// TIA Portal V16 export
// export: Created 2021-03-19T14:27:15.418879Z, ExportSetting WithDefaults, DisplayName Totally Integrated Automation Portal, DisplayVersion V16 Update 3, DisplayName TIA Portal Version Control Interface, DisplayVersion V16 Update 2, DisplayName TIA Portal Openness, DisplayVersion V16 Update 3, DisplayName STEP 7 Professional, DisplayVersion V16 Update 3, DisplayName STEP 7 Safety, DisplayVersion V16, DisplayName WinCC Professional, DisplayVersion V16 Update 3
FUNCTION "FC02001_StdInstAnalogRead" : Void   // FC2001, LAD
TITLE = Standard - Inst — Analog Instrument Read and Scale
{ S7_Optimized_Access := 'TRUE' }
AUTHOR : M_Gledhill
FAMILY : Instrumentation
NAME : StdInstAnalogRead
VERSION : 1.0
// PRACTICAL SERIES AUTOMATION LIBRARY (PAL)   —   COPYRIGHT 2020 – M. GLEDHILL (MIT LICENCE)
//                   ———— ◆ ————
//  FOR DETAILED DOCUMENTATION — SELECT THE BLOCK IN THE PROJECT TREE AND PRESS SHIFT + F1
//  FULL ONLINE DOCUMENTATION IS AVAILABLE AT: https://practicalseries.com/2001-pal/index.html
// stored: AutoNumber false, IsIECCheckEnabled false, SetENOAutomatically false, UDAEnableTagReadback false
   VAR_INPUT
      SYS_SIGNALS : "UT21000_Dy_SysSignals";   // Common system signals — logic and timing signals
      RAW_ANALOG : Int;   // Analogue Input Signal
      EXT_FAULT : Bool;   // Instrument External Fault (1 = Fault, 0 = Healthy)
   END_VAR
   VAR_IN_OUT
      STATIC_DATA : "UT02001_St_InstAnalogRead";   // Static data storage (UDT)
      DYNAMIC_DATA : "UT22001_Dy_InstAnalogRead";   // Dynamic data storage (UDT)
   END_VAR
   VAR_TEMP
      revInfo : "UT01000_St_SysRevision";   // Revision information for this block
      licInfo : "UT01001_St_SysLicence";   // Licence information for this block
      wrkAlmHEn : Bool;   // Working storage (Alm_H is enabled and not masked)
      wrkAlmLEn : Bool;   // Working storage (Alm_L is enabled and not masked)
      wrkWrnHEn : Bool;   // Working storage (Wrn_H is enabled and not masked)
      wrkWrnLEn : Bool;   // Working storage (Wrn_L is enabled and not masked)
      calcPart1 : Real;   // Scale value calculation part 1 (RAW_VALUE − RAW_MIN)
      calcPart2 : Real;   // Scale value calculation part 2 (SCALE_MAX − SCALE_MIN)
      calcPart3 : Real;   // Scale value calculation part 1 (RAW_MAX − RAW_MIN)
      calcRawOOR : Real;   // Calculated OOR absolute value in terms of the RAW_VALUE
      calcOverRange : Real;   // Calculated over range limit (in raw units)
      calcUnderRange : Real;   // Calculated under range limit (in raw units)
      calcHystAbs : Real;   // Absolute Hysteresis (in relation to alarm/waringin)
      wrkHyst : Real;   // Working hysteresis value
      wrkOORPercent : Real;   // Working out of range percentage
      wrkInt : Int;   // Working storage (Integer)
      wrkReal : Real;   // Working storage (real)
      wrkDInt : DInt;   // Working storage (Double integer)
   END_VAR
   VAR_TEMP   // added for the SCL form of the ladder/FBD networks
      _w1 : Bool;
      _w2 : Bool;
      _w3 : Bool;
      _w4 : Bool;
   END_VAR
BEGIN

REGION Network 1: Block description — Sections 1 to 3.1
   // ▀▀▀▀▀▀▀▀▀▀▀▀▀▀▀▀▀▀▀▀▀▀▀▀▀▀▀▀▀▀▀▀▀▀▀▀▀▀▀▀▀▀▀▀
   // 
   // TITLE:    STANDARD ANALOG INSTRUMENT READ, SCALE AND ALARM MONITORING
   // 
   // ▄▄▄▄▄▄▄▄▄▄▄▄▄▄▄▄▄▄▄▄▄▄▄▄▄▄▄▄▄▄▄▄▄▄▄▄▄▄▄▄▄▄▄▄
   // 
   // 
   // 
   // This block reads and scales an analogue instrument signal received via an analogue input card.
   // 
   // The resultant scaled value is a real (floating point) number that matches the calibrated range of 
   // the instrument in engineering units.
   // 
   // The block has the facility to generate up to four alarms and warnings whenever the signal is 
   // beyond a specific setpoint value (either above or below); the four signals are:
   // 
   //    •   Alarm high
   // 
   //    •   Warning high
   // 
   //    •   Warning low
   // 
   //    •   Alarm low
   // 
   // Each alarm or warning can be time filtered (the condition must be present for a preset time 
   // before the alarm or warning is activated) and each will automatically reset when the signal is 
   // back within the acceptable range by a hysteresis amount.
   // 
   // In addition to the above four signals, various out-of-range fault signals will be generated if the 
   // instrument is outside its normal calibrated range by more than a specified percentage (this 
   // being a percentage of the total span of the instruments range).
   // 
   // The block can also generate an optional “external fault” signal from a hardwired fault input from 
   // the instrument itself.
   // 
   // The block has a simulation mode whereby the scaled value is replaced by an operator selected 
   // value (over-writing any signal from the instrument). This can be used for testing purposes or if 
   // the instrument is out of service for any reason.
   // 
   // 
   // 
   // 
   // 
   // ▄▄▄▄▄▄▄▄▄▄▄▄▄▄▄▄▄▄▄▄▄▄▄▄▄▄▄▄▄▄▄▄▄▄▄▄▄▄▄▄▄▄▄▄
   // 1.     BLOCK TECHNICAL SUMMARY
   // 
   // 
   //  ――――――――――――――――――――――――――――――――――――――――――
   //  NOMENCLATURE & ADDRESSING
   //  ――――――――――――――――――――――――――――――――――――――――――
   //  BLOCK TITLE         Analog Instrument Read, Scale and Alarm Monitoring
   //  BLOCK FUNCTION GROUP    Instrument 
   //  BLOCK ADDRESS       FC02001
   //  BLOCK SYMBOL        FC02001_StdInstAnalogRead
   //  BLOCK USER ID         StdInstAnalogRead
   // 
   //  ――――――――――――――――――――――――――――――――――――――――――
   //  BLOCK TYPE & USAGE
   //  ――――――――――――――――――――――――――――――――――――――――――
   //  BLOCK TYPE         Function (FC)
   //  BLOCK NUMBER        02001
   //  LANGUAGE           LAD
   //  OPTIMISED ACCESS     Yes
   //  PAL USAGE TYPE       Standard block
   // 
   //  ――――――――――――――――――――――――――――――――――――――――――
   //  METRICS
   //  ――――――――――――――――――――――――――――――――――――――――――
   //  EXECUTION TIME       87.69 μs¹
   //  LOAD MEMORY       83.17 kB  (85171 bytes)
   //  WORK MEMORY           2.16 kB    (2215 bytes)
   //  ――――――――――――――――――――――――――――――――――――――――――
   //                ¹ Measured on: CPU-1515-2PN/DP (order no. 6ES7 515-2AM02-0AB0)
   // 
   //                ━━━   ⬙⬙⬙⬙⬙⬙   ━━━
   // 
   // 
   // 
   // ▄▄▄▄▄▄▄▄▄▄▄▄▄▄▄▄▄▄▄▄▄▄▄▄▄▄▄▄▄▄▄▄▄▄▄▄▄▄▄▄▄▄▄▄
   // 2.     FUNCTIONAL DESCRIPTION
   // 
   // This block is a comprehensive block designed to read and scale an analogue instrument; it 
   // provides the following broad functions:
   // 
   //    •   Read an analogue input, convert it to a real number that represents the calibrated 
   //      range of the instrument in engineering units
   // 
   //    •   Generate high and low alarm and warning signals to indicate that the instrument is 
   //      above or below specific thresholds
   // 
   //    •   Generate fault signals if the instrument is out of range or is indicating a specific fault 
   //      condition
   // 
   //    •   Provide simulation capabilities for testing and fault handling situations
   // 
   //    •   Generates the status and message signals necessary for symbolic representation at 
   //      a supervisory system (SCADA or HMI)
   // 
   // 
   // 
   // ▂▂▂▂▂▂▂▂▂▂▂▂▂▂▂▂▂▂▂▂▂▂▂▂▂▂▂▂▂▂▂▂▂▂▂▂▂▂▂▂▂▂▂▂
   // 2.1     Read and scale and instrument signal
   // 
   // The principal function of the block is to read a raw integer signal from an analogue instrument 
   // (in the form of an input word, IW), and convert it into a scaled, floating point (real) number that 
   // reflects the calibrated reading of the instrument in question.
   // 
   // For example, if a flow meter with a calibrated range of -100 l/s to +100 l/s provided a 4-20 mA 
   // signal to the PLC, then 4 mA would represent -100 l/s and 20 mA would rep-resent +100 l/s.
   // 
   // A typical 4-20 mA analogue input signal returns raw value of 0 at 4 mA and 27648 at 20 mA. 
   // 
   // The block would return scaled values as follows (it would also return every value in between; five 
   // typical values have been shown):
   // 
   // 
   //  ――――――――――――――――――――――――――――――――――――――――――
   //  RAW_SIGNAL          RAW INTEGER VALUE        RETURNED SCALE VALUE
   //  ――――――――――――――――――――――――――――――――――――――――――
   //     4 mA                      0             -100 l/s
   //     8 mA               6912                   -50 l/s
   //   12 mA             13824                   0 l/s
   //   16 mA             20736              +50 l/s
   //   20 mA             27648            +100 l/s
   //  ――――――――――――――――――――――――――――――――――――――――――
   // 
   // 
   // 
   // ▂▂▂▂▂▂▂▂▂▂▂▂▂▂▂▂▂▂▂▂▂▂▂▂▂▂▂▂▂▂▂▂▂▂▂▂▂▂▂▂▂▂▂▂
   // 2.2     Alarms and warnings
   // 
   // 
   // The block provides four alarm/warning signals:
   // 
   // 
   //  ――――――――――――――――――――――――――――――――――――――――――
   //  ALARM/WARNING         FUNCTION
   //  ――――――――――――――――――――――――――――――――――――――――――
   //  Alarm high            Scaled signal is equal to or above a preset alarm high 
   //                threshold (setpoint)
   // 
   //  Warning high           Scaled signal is equal to or above a preset warning high
   //                threshold (setpoint)
   // 
   //  Warning low          Scaled signal is equal to or above a preset warning low
   //                threshold (setpoint)
   // 
   //  Alarm low              Scaled signal is equal to or above a preset alarm low
   //                threshold (setpoint)
   //  ――――――――――――――――――――――――――――――――――――――――――
   // 
   // 
   // Alarms and warnings are individually enabled and are individually configurable.
   // 
   // Each alarm or warning has a threshold value (the value at which it becomes active); high alarms 
   // and warnings are active when the instrument is at or above the threshold level, low alarms and 
   // warnings are active when the instrument is at or below the threshold level. 
   // 
   // Each alarm or warning also has a hysteresis value (the instrument must be inside the threshold 
   // value by at least the hysteresis amount before the alarm/warning is reset).
   // 
   // Alarms and warnings automatically reset once the instrument is inside the threshold value by at 
   // least the hysteresis value.
   // 
   // Each alarm or warning is equipped with on and off time filtering (to prevent nuisance triggering 
   // of alarms and warnings) where:
   // 
   // ON FILTERING:  Delays the activation of the alarm/warning (signal must
   //          be on for a time period before the block conditioned 
   //          signal is activated).
   // 
   // OFF FILTERING:    Delays the alarm/warning from going off (i.e. the 
   //          conditioned signal will remain on for a time period
   //          once the input is reset).
   // 
   // Each alarm and warning has its own configurable on and off filtering delays.
   // 
   // 
   // 
   // ▂▂▂▂▂▂▂▂▂▂▂▂▂▂▂▂▂▂▂▂▂▂▂▂▂▂▂▂▂▂▂▂▂▂▂▂▂▂▂▂▂▂▂▂
   // 2.3     Fault signals
   // 
   // The block is able to generate four fault signals:
   // 
   //    •   External fault
   //    •   Instrument is over-range
   //    •   Instrument is under-range
   //    •   Instrument is out-of-range (common signal)
   // 
   // The external fault is generated by a hardwired signal from the instrument that indicates the 
   // instrument itself is reporting a fault. External fault signals are common with certain types of 
   // instrument (mass flow meters &c.) and are used to indicate such things as medium not present 
   // (liquid flow meters) or calibration and maintenance issues (instrument requires calibrating or 
   // cleaning or some other form of servicing).
   // 
   // Over-range and under-range faults are generated if the instrument is reading outside its normal 
   // calibrated range. Over-range if the instrument is reading higher than its maximum permitted 
   // value and under-range if lower than its minimum permitted value.
   // 
   // The level at which the instrument is considered to be either over-range or under-range (out of 
   // range), is set as a percentage of the whole instrument range (the span or full-scale deflection).
   //  
   // In the example of § 2.1, the instrument had a range of -100 to +100 l/s, this is a total range of 
   // 200 l/s, if the out of range value were set at 2.5%, this would be 2.5% of 200 l/s or 5 l/s. Thus, the 
   // instrument would be over-range if it were reading above 105 l/s; it would be under-range below
   // -105 l/s.
   // 
   // The out-of-range fault signal is a common signal the activates if either the over-range or 
   // under-range signal is active. It indicated the instrument is either over-range or under-range, but 
   // doesn’t specify which.
   // 
   // 
   // 
   // ▂▂▂▂▂▂▂▂▂▂▂▂▂▂▂▂▂▂▂▂▂▂▂▂▂▂▂▂▂▂▂▂▂▂▂▂▂▂▂▂▂▂▂▂
   // 2.4     Operating modes
   // 
   // The block supports the following optional modes of operation:
   // 
   //    •   Simulation mode (allows the operator to override the current instrument reading 
   //      with a simulated value)
   // 
   //    •   Remote/local/all selection (allows control of the instrument to be restricted to a 
   //      specific SCADA/HMI device) 
   // 
   //    •   Faceplate disabled (disables all optional modes)
   // 
   // 
   // 
   // ▁▁▁▁▁▁▁▁▁▁▁▁▁▁▁▁▁▁▁▁▁▁▁▁▁▁▁▁▁▁▁▁▁▁▁▁▁▁▁▁▁▁▁▁
   // 2.4.1     Simulation mode
   // 
   // The instrument can be switched to a simulation mode, in which the actual reading from the 
   // instrument is replaced by a simulated value provided by the operator. Simulation mode can be 
   // used during testing and can also be applied in a process environment if a fault condition is 
   // detected within the instrument.
   // 
   // Simulation mode is a manual operation that can only be initiated by an operator.
   // 
   // 
   // 
   // ▁▁▁▁▁▁▁▁▁▁▁▁▁▁▁▁▁▁▁▁▁▁▁▁▁▁▁▁▁▁▁▁▁▁▁▁▁▁▁▁▁▁▁▁
   // 2.4.2     Remote/local/all mode
   // 
   // Remote and local operating modes refer to the device that has control of the instrument; where 
   // a plant has more than one SCADA/HMI, say a SCADA in a remote control room and a field 
   // mounted HMI local to the instrument, it is possible to restrict the control of the instrument to 
   // one, or the other, or both devices as follows:
   // 
   //    •   Remote Only the remote system in the control room can control the 
   // 
   //    •   Local     A local system has taken control of the device and the remote system can 
   //            no longer issue commands to it
   // 
   //    •    All    Any system can control the device
   // 
   // The default arrangement if for all system to have access to the device.
   // 
   // 
   // 
   // ▁▁▁▁▁▁▁▁▁▁▁▁▁▁▁▁▁▁▁▁▁▁▁▁▁▁▁▁▁▁▁▁▁▁▁▁▁▁▁▁▁▁▁▁
   // 2.4.3     Facepalte disabled mode
   // 
   // Prevents the supervisory system from displaying the faceplate from which the above options are 
   // selected. If the faceplate is disabled, this module will set re-mote/local mode to ALL and will 
   // disable simulation mode.
   // 
   // 
   // 
   // ▁▁▁▁▁▁▁▁▁▁▁▁▁▁▁▁▁▁▁▁▁▁▁▁▁▁▁▁▁▁▁▁▁▁▁▁▁▁▁▁▁▁▁▁
   // 2.4      Supervisory system interface
   // 
   // See the online documentation for this block — select the block in the project tree and press:
   //      SHIFT + F1
   // 
   // The supervisory system interface is available in section 2.5 of the online SMDS document.
   // 
   //                ━━━   ⬙⬙⬙⬙⬙⬙   ━━━
   // 
   // 
   // 
   // ▄▄▄▄▄▄▄▄▄▄▄▄▄▄▄▄▄▄▄▄▄▄▄▄▄▄▄▄▄▄▄▄▄▄▄▄▄▄▄▄▄▄▄▄
   // 3.     DETAILED BLOCK DESCRIPTION
   // 
   // This block, FC02001_StdInstAnalogRead uses user data types to provide the primary interface 
   // to the block. There are five formal parameters: 
   // 
   //  ――――――――――――――――――――――――――――――――――――――――――
   //  PARAM         FUNCTION                    TYPE      IN-OUT 
   //  ――――――――――――――――――――――――――――――――――――――――――
   //  SYS_SIGNALS      Common system signals              UT21000    In
   //           logic and timing signals for parametric access
   // 
   //  RAW_ANALOG      The unscaled analogue input (input word        Word     In
   //           address for the IO card to which the instrument 
   //           is connected)
   // 
   //  EXT_FAULT     Optional external fault signal for the instrument     Bool      In
   //           (1 = fault, 0 = healthy). If not required, set 
   //           permanently to _False
   // 
   //  STATIC_DATA     Data structure that holds the configuration data    UT02001    In
   //           for the instrument (raw range, scaled range 
   //           alarm and warning values, filtering times, 
   //           hysteresis values &c.)
   // 
   //  DYNAMIC_DATA      Data structure that holds the live data for the      UT22001    InOut
   //           instrument (its reading in engineering units, 
   //           any alarms or warnings that may be active, 
   //           current timer values, selected operating 
   //           mode &c.)
   //  ――――――――――――――――――――――――――――――――――――――――――
   // 
   // RAW_ANALOG and EXT_FAULT are signals provided directly from the instrument itself (via input 
   // cards). The other two parameters: STATIC_DATA and DYNAMIC_DATA are UDTs that hold 
   // (respectively) the configuration information and the live data for the instrument.
   // 
   //  ――――――――――――――――――――――――――――――――――――――――――
   //  PARAM         ASSOCIATED UDT            ASSOCIATED DATA BLOCK
   //  ――――――――――――――――――――――――――――――――――――――――――
   //  STATIC_DATA     UT02001_St_InstAnalogRead     DB02001_St_InstAnalogRead
   //  DYNAMIC_DATA      UT22001_Dy_InstAnalogRead       DB22001_Dy_InstAnalogRead
   //  ――――――――――――――――――――――――――――――――――――――――――
   // 
   // Section 5 contains a full list of all variables within these UDTs.
   // 
   // This arrangement conforms with the PAL philosophy whereby IO card connections have unique 
   // formal parameters; all remaining signals are passed as variables within UDTs.
   // 
   // 
   // 
   // ▂▂▂▂▂▂▂▂▂▂▂▂▂▂▂▂▂▂▂▂▂▂▂▂▂▂▂▂▂▂▂▂▂▂▂▂▂▂▂▂▂▂▂▂
   // 3.1     Converting the raw instrument signal to a scaled value
   // 
   // The RAW_ANALOG is the raw instrument signal received from an analogue input card; these have 
   // specific ranges depending on the type of IO card and the type of signal in use.
   //  
   // Note:    It is assumed that the instrument has a linear response.
   // 
   // The following tables show the typical ranges for the RAW_ANALOG:
   // 
   // 
   //  ――――――――――――――――――――――――――――――――――――――――――
   //             LOWER LIMIT     EQUIVALENT   UPPER LIMIT     EQUIVALENT
   //  SIGNAL TYPE      (RAW_MIN)          TO      (RAW_MAX)         TO
   //  ――――――――――――――――――――――――――――――――――――――――――
   //  -10 V to 10 V         -27648      -10 V          27648        +10 V
   //  -5 V to 5 V       -27648        -5 V          27648       +5 V
   //  -2.5 V to 2.5 V       -27648        -2.5 V          27648       +2.5 V
   //  -1 V to 1 V       -27648        -1 V          27648       +1 V
   //  -500 mV to 500 mV      -27648       -500 mV      27648      +500 mV
   //  -250 mV to 250 mV      -27648       -250 mV      27648      +250 mV
   //  -80 mV to 80 mV       -27648      -80 mV      27648        +80 mV
   //  -50 mV to 50 mV    -27648      -50 mV      27648        +50 mV
   //  1 V to 5 V          0       +1 V          27648       +5 V
   //  ――――――――――――――――――――――――――――――――――――――――――
   //  Input ranges for typical instrument types (voltage)
   // 
   // 
   // 
   //  ――――――――――――――――――――――――――――――――――――――――――
   //             LOWER LIMIT     EQUIVALENT   UPPER LIMIT     EQUIVALENT
   //  SIGNAL TYPE      (RAW_MIN)          TO      (RAW_MAX)         TO
   //  ――――――――――――――――――――――――――――――――――――――――――
   //  -500 mV to 500 mV   -27648       -500 mV      27648      +500 mV
   //  -20 mA to 20 mA       -27648      -20 mA      27648        +20 mA
   //  0 mA to 20 mA         0         0 mA      27648        +20 mA
   //  4 mA to 20 mA         0         4 mA      27648        +20 mA
   //  ――――――――――――――――――――――――――――――――――――――――――
   //  Input ranges for typical instrument types (current)
   // 
   // 
   // 
   // 
   //  ――――――――――――――――――――――――――――――――――――――――――
   //             LOWER LIMIT     EQUIVALENT   UPPER LIMIT     EQUIVALENT
   //  SIGNAL TYPE      (RAW_MIN)          TO      (RAW_MAX)         TO
   //  ――――――――――――――――――――――――――――――――――――――――――
   //  RTD 150 Ω            0         0 Ω         27648        150 Ω
   //  RTD 300 Ω            0         0 Ω         27648        300 Ω
   //  RTD 600 Ω            0         0 Ω         27648        600 Ω
   //  RTD 6000 Ω         0         0 Ω         27648      6000 Ω
   //  PT x00           -2000        200.0°C        8500        850.0°C
   //  Ni x00          -600      -60.0°C          250        250.0°C
   //  Type B thermocouple     -2100       -210.0°C        12000      1200.0°C
   //  Type K thermocouple     -2700       -270.0°C        13720      1372.0°C
   //  Type N thermocouple    -2700       -210.0°C        13000      1300.0°C
   //  Type R/S thermocouple    -500      -50.0°C        17690      1769.0°C
   //  Type T thermocouple     -2700       -270.0°C        4000        400.0°C
   //  ――――――――――――――――――――――――――――――――――――――――――
   //  Input ranges for typical instrument types (resistance thermometers and thermocouples)
   // 
   // The RAW_MIN and the RAW_MAX values in the above tables are the numerical values for the 
   // instrument range; the appropriate values must be entered in the STATIC_DATA data structure 
   // passed to the block. These are the UDT variables:
   // 
   //  UT02001_St_InstAnalogRead
   //  ――――――――――――――――――――――――――――――――――――――――――
   //  SIGNAL NAME          FUNCTION                     TYPE
   //  ――――――――――――――――――――――――――――――――――――――――――
   //  RANGE_RAW_MIN       RANGE — Minimum value of the raw analogue    Int
   //                     signal (at the card)
   //  RANGE_RAW_MAX      RANGE — Maximum value of the raw analogue      Int
   //                     signal (at the card)
   //  ――――――――――――――――――――――――――――――――――――――――――
   // 
   // The corresponding values for the scaled instrument signal are:
   // 
   //  UT02001_St_InstAnalogRead
   //  ――――――――――――――――――――――――――――――――――――――――――
   //  SIGNAL NAME          FUNCTION                     TYPE
   //  ――――――――――――――――――――――――――――――――――――――――――
   //  RANGE_SCALE_MIN      RANGE — Minimum value of the scaled analogue     Real
   //                     signal [engineering units]
   //  RANGE_SCALE_MAX     RANGE — Maximum value of the scaled analogue    Real
   //                     signal [engineering units]
   //  ――――――――――――――――――――――――――――――――――――――――――
   // 
   // Thus, if a flow meter with a calibrated range of -100 l/s to +100 l/s provided a 4 20 mA signal to 
   // the PLC, then:
   // 
   //  ――――――――――――――――――――――――――――――――――――――――――
   //  RANGE_RAW_MIN   RANGE_RAW_MAX   RANGE_SCALE_MIN     RANGE_SCALE_MAX
   //  ――――――――――――――――――――――――――――――――――――――――――
   //         0           27648             -100.0            +100.0
   //  ――――――――――――――――――――――――――――――――――――――――――
   // 
   // The scaled value is stored in the DATA_DYNAMIC structure in the following variable:
   // 
   //  UT22001_Dy_InstAnalogRead
   //  ――――――――――――――――――――――――――――――――――――――――――
   //  SIGNAL NAME          FUNCTION                     TYPE
   //  ――――――――――――――――――――――――――――――――――――――――――
   //  actual_Value          ACTUAL — SCALED INSTRUMENT VALUE         Real
   //                      [engineering units]
   //  ――――――――――――――――――――――――――――――――――――――――――
   // 
   // The scaled value (actual_Value) is calculated as follows:
   // 
   // 
   // ┌─────────────────────────────────────────┐
   // │                              (RAW_ANALOG ─ RAW_MIN) ╳ (SCALE_MAX ─ SCALE_MIN)            │
   // │actual_Value =  ――――――――――――――――――――――――――  ┼ SCALE_MIN    │
   // │                              (RAW_MAX ─ RAW_MIN)                    │
   // └───────────────────────────────────  (3.1)  ───┘
   // Note:    RAW_MIN, RAW_MAX,  SCALE_MIN and SCALE_MAX are all preceded with RANGE_
   //      in the above equation 
   // 
   // 
   // 
   //            SCALE_VALUE
   //             ↑                    ⋰
   //    RANGE_SCALE_MAX__│______________________________________⋰
   //             │                  ╱|
   //             │                 ╱ |     
   //             │                ╱  |
   //             │               ╱   |
   //             │              ╱    |
   //             │             ╱     |
   //             │            ╱      |
   //         actual_Value │<- - - - - - - - - - - - - - - - - - - - - ╱       |
   //             │          ╱ ⌃           |
   //             │         ╱ ╎       |
   //             │        ╱  ╎       |
   //             │       ╱   ╎       |   
   //             │      ╱    ╎       |
   //             │     ╱     ╎       |
   //             │    ╱         ╎          |
   //     RANGE_SCALE_MIN__│______╱          ╎          |
   //             │  ⋰|           ╎          |
   //             │ ⋰ |           ╎          |
   //             ┼─────────────────────────→ RAW_ANALOG
   //                   |           ╎           |
   //             RANGE_RAW_MIN      ╎     RANGE_RAW_MAX
   //                        RAW_ANALOG
   // 
   //            Linear relationship between RAW_ANALOG and actual_Value
   // 
   // 
   // 
   // ▁▁▁▁▁▁▁▁▁▁▁▁▁▁▁▁▁▁▁▁▁▁▁▁▁▁▁▁▁▁▁▁▁▁▁▁▁▁▁▁▁▁▁▁
   // 3.1.1     Configuration errors
   // 
   // The block requires that both the RANGE_RAW and RANGE_SCALE signals conform to certain rules:
   // 
   //    1.  RANGE_RAW_MIN must be less than, and not equal to RANGE_RAW_MAX
   //    2.  RANGE_SCALE_MIN must be less than, and not equal to RANGE_SCALE_MAX
   // 
   // Should either of these conditions not be met, the signal: status_ConfigError will be activated 
   // (set true), additionally the three out of range signals (see § 3.3.1):
   // 
   //      msg_Flt_OverRange
   //      msg_Flt_UnderRange
   //      msg_Flt_OutOfRange
   // 
   // Will all be activated (this condition cannot be over-ridden by simulation mode, see § 3.4.1) and 
   // the actual_Value will be set to zero irrespective of any values given to RAW_ANALOG.
   // 
   // Note:    This avoids the potential for a divide by zero error: if the RANGE_RAW_MIN and 
   //      RANGE_RAW_MAX are exactly equal, the calculation of the actual_Value in 
   //      equation (3.1) would result in a divide by zero error.
END_REGION

REGION Network 2: Block description — Sections 3.2 to 3.7
   // ▂▂▂▂▂▂▂▂▂▂▂▂▂▂▂▂▂▂▂▂▂▂▂▂▂▂▂▂▂▂▂▂▂▂▂▂▂▂▂▂▂▂▂▂
   // 3.2     Warnings and alarms
   // 
   // By default, the block generates 4 alarms and warnings (2 warnings and 2 alarms, 4 in total) 
   // as follows:
   // 
   // 
   //  ――――――――――――――――――――――――――――――――――――――――――
   //  ALARM / WARNING     FUNCTION
   //  ――――――――――――――――――――――――――――――――――――――――――
   //  Alarm high       Scaled signal is equal to or above a preset alarm high setpoint
   //  Warning high      Scaled signal is equal to or above a preset warning high setpoint
   //  Warning low     Scaled signal is equal to or below a preset warning low setpoint
   //  Alarm low      Scaled signal is equal to or below a preset alarm low setpoint
   //  ――――――――――――――――――――――――――――――――――――――――――
   //  Default alarm and warning signals
   // 
   // 
   // The active state of any alarm or warning is stored in the DATA_DYNAMIC structure in the following 
   // variables:
   // 
   //  UT22001_Dy_InstAnalogRead
   //  ――――――――――――――――――――――――――――――――――――――――――
   //  SIGNAL NAME          FUNCTION                     TYPE
   //  ――――――――――――――――――――――――――――――――――――――――――
   //  msg_Alm_H         MESSAGE — Alarm - high alarm is active        Bool
   //  msg_Alm_L          MESSAGE — Alarm - low alarm is active          Bool
   //  msg_Wrn_H          MESSAGE — Warning - high warning is active      Bool
   //  msg_Wrn_L          MESSAGE — Warning - low warning is active        Bool
   //  ――――――――――――――――――――――――――――――――――――――――――
   // 
   // The alarms and warnings that end with _H are activated when the scaled instrument reading is 
   // greater than or equal to a setpoint threshold (i.e. activate when the measured quantity is too 
   // high; generally, if there is both an alarm high and a warning high, the convention within the PAL 
   // is that the warning should activate before the alarm².
   // 
   // 
   // The alarms and warnings that end with _L are activated when the scaled instrument reading is 
   // less than or equal to a setpoint threshold (i.e. activate when the measured quantity is too high; 
   // generally, if there is both an alarm low and a warning low, the convention within the PAL is that 
   // the warning should activate before the alarm².
   // 
   // ――――――――――
   // ²         This is just a convention, there is nothing to stop the warning being set to occur after 
   //      the alarm (i.e. the warning detecting the most extreme condition). All alarms and 
   //      warnings are entirely independent of each other and no error checking is carried 
   //      out to ensure that any particular threshold is above or below another.
   // ――――――――――
   // 
   // All alarms and warnings are individually enabled (a disabled alarm or warning will never be 
   // activated), all alarms and warnings have individual setpoint values (the value at which the 
   // alarm or warning is triggered), all alarms and warnings have individual hysteresis valves 
   // (effectively a tolerance band, the difference between where an alarm activates and where is 
   // deactivates, used to prevent nuisance or “chattering” alarms). Finally, each alarm and warning 
   // has a configurable on and off delay (the alarm or warning will only activate if the reading is 
   // outside the threshold for the on-delay time and similarly will only deactivate when the reading 
   // is inside the threshold and hysteresis for the off-delay time).
   // 
   // The following table summarises all the available signals for each alarm and warning:
   // 
   //  ――――――――――――――――――――――――――――――――――――――――――
   //  SIGNAL          FUNCTION             TYPE   DETAILS
   //  ――――――――――――――――――――――――――――――――――――――――――
   //  CONFIG_XXX_Y_ENABLE Alarm/warning enabled      Bool    1 = enabled, 0 = disabled
   //  SP_XXX_Y_VAL      Alarm/warning setpoint value    Real Engineering units
   //  SP_XXX_Y_HYST_VAL    Alarm/warning hysteresis value Real Engineering units
   //  TIME_XXX_Y_ON_DEL   Alarm/warning on delay time   Real In seconds
   //  TIME_XXX_Y_OFF_DEL     Alarm/warning off delay time   Real In seconds
   //  mode_Xxx_Y_MaskOn     Alarm/warning is masked      Bool    1 = masked, 0 = normal
   //  msg_Xxx_Y         Alarm/warning is active      Bool    1 = active, 0 = inactive
   //  ――――――――――――――――――――――――――――――――――――――――――
   //  Default alarm and warning signals — where XXX is either ALM or WRN and Y is either H or L
   // 
   // 
   // 
   // ▁▁▁▁▁▁▁▁▁▁▁▁▁▁▁▁▁▁▁▁▁▁▁▁▁▁▁▁▁▁▁▁▁▁▁▁▁▁▁▁▁▁▁▁
   // 3.2.1     High alarms and warnings (an example)
   // 
   // This example explains how a high alarm signal is generated, a high warning works in exactly the 
   // same way with WRN being substituted for ALM.
   // 
   // The full set of signals associated with the high alarm are:
   // 
   //  ――――――――――――――――――――――――――――――――――――――――――
   //  SIGNAL           FUNCTION            TYPE   DETAILS
   //  ――――――――――――――――――――――――――――――――――――――――――
   //  SP_ALM_H_VAL      Alarm high setpoint value    Real Engineering units
   //  SP_ALM_H_HYST_VAL    Alarm high hysteresis value Real Engineering units
   //  TIME_ALM_H_ON_DEL   Alarm high on delay time   Real In seconds
   //  TIME_ALM_H_OFF_DEL     Alarm high off delay time   Real In seconds
   //  mode_Alm_H_MaskOn    Alarm is masked         Bool    1 = masked, 0 = normal
   //  msg_Alm_H        Alarm high is active      Bool    1 = active, 0 = inactive
   //  ――――――――――――――――――――――――――――――――――――――――――
   // 
   // The figure below indicates how each of these signal functions (note TIME_ALM_H_ON_DEL and
   // TIME_ALM_H_OFF_DEL have been abbreviated to ON_DEL and OFF_DEL respectively):
   // 
   // 
   //                 │
   //                 │          ╱╲╱╲
   //                 │    ①      ②╱    ╲
   //       SP_ALM_H_VAL↘│____╱╲________╱____________╲③_______④__________ 
   //    SP_ALM_H_HYST_VAL ↕│__╱____╲____╱╎_____╎_______╲____╱╲___________
   //                 │╱    ╲╱ ╎    ╎      ╲╱     ╲
   //                 │        ╎    ╎          ╎╲
   //                 │        ╎    ╎          ╎ ╲___
   //                 │        ╎    ╎          ╎    ╎╲╱
   //                 │    ON_DEL→╎    ╎←    OFF_DEL→╎    ╎←
   //                 ┼─────────────────────────────
   // 
   //                            ╎                        ╎
   // 
   //         msg_Alm_H │             ┏━━━━━━━━━━━━┓
   //                 │             ┃               ┃
   // CONFIG_ALM_H_ENABLE = 1  │             ┃   ALARM IS ACTIVE    ┃
   // & mode_Alm_H_MaskOn = 0 │             ┃               ┃
   //                 │             ┃               ┃
   //                 ┼━━━━━━━━━━━━╶╶╶╶╶╶╶╶╶╶╶╶╶━━━━
   // 
   //                            ╎                        ╎
   // 
   //         msg_Alm_H │          
   // ⑤               │             ╎               ╎             
   // CONFIG_ALM_H_ENABLE = 0  │             
   //     OR          │             ╎               ╎
   // CONFIG_ALM_H_ENABLE = 1  │          
   // & mode_Alm_H_MaskOn = 1 ┼━━━━━━━━━━━━━━━━━━━━━━━━━━━━━
   // 
   // 
   // 
   // ▁▁▁▁▁▁▁▁▁▁▁▁▁▁▁▁▁▁▁▁▁▁▁▁▁▁▁▁▁▁▁▁▁▁▁▁▁▁▁▁▁▁▁▁
   // Scenario ①, alarm setpoint reached, but for less than on-delay duration
   // 
   // The graph represents the scaled analogue instrument reading, actual_Value (in engineering 
   // units). The top horizontal line is the setpoint for the high alarm (SP_ALM_H_VAL).
   // 
   // If the alarm is enabled (CONFIG_ALM_H_ENABLE = 1) then the following actions occur:
   // 
   // At point ① on the graph, the signal actual_Value reaches (and exceeds) the threshold value 
   // SP_ALM_H_VAL; i.e.:
   // 
   //           actual_Value ≥ SP_ALM_H_VAL
   // 
   // At this point, the alarm setpoint is exceeded and the on-delay timer starts; in the case of point ①, 
   // the signal actual_Value falls back below the setpoint value before the on-delay timer reaches 
   // the time set in TIME_ALM_H_ON_DEL, consequently the alarm does not activate.
   // 
   // 
   // 
   // ▁▁▁▁▁▁▁▁▁▁▁▁▁▁▁▁▁▁▁▁▁▁▁▁▁▁▁▁▁▁▁▁▁▁▁▁▁▁▁▁▁▁▁▁
   // Scenario ②, alarm setpoint reached for more than the on-delay duration
   // 
   // At point ② on the graph, the signal actual_Value again reaches (and exceeds) the setpoint value 
   // SP_ALM_H_VAL.
   // 
   // Again, at this point, the alarm threshold is exceeded and the on-delay timer starts; in the case of 
   // point ②, the signal actual_Value remains at or above the setpoint value for the full duration of 
   // the TIME_ALM_H_ON_DEL and consequently the alarm activates (msg_Alm_H goes to a high 
   // state), this is indicated in the middle msg_Alm_H graph.
   // 
   // 
   // 
   // ▁▁▁▁▁▁▁▁▁▁▁▁▁▁▁▁▁▁▁▁▁▁▁▁▁▁▁▁▁▁▁▁▁▁▁▁▁▁▁▁▁▁▁▁
   // Scenario ③, alarm reset level reached, but for less than the off-delay duration
   // 
   // At point ③, the signal actual_Value falls to the point at which the alarm is no longer active i.e.:
   // 
   //           actual_Value < (SP_ALM_H_VAL − SP_ALM_H_HYST_VAL)
   // 
   // Note:    in this case the inequality is less than (not less than or equal to), this is to prevent 
   //      conflict detecting the threshold and detecting the reset value if SP_ALM_H_HYST_VAL 
   //      is set to zero.
   // 
   // At this point, the signal is below the alarm reset level:
   // 
   //           SP_ALM_H_VAL − SP_ALM_H_HYST_VAL
   // 
   // and the off-delay timer starts; in the case of point 3, the signal actual_Value re-turns above the 
   // reset threshold before the off-delay timer reaches the time set in TIME_ALM_H_OFF_DEL, 
   // consequently, the alarm does not deactivate.
   // 
   // 
   // 
   // ▁▁▁▁▁▁▁▁▁▁▁▁▁▁▁▁▁▁▁▁▁▁▁▁▁▁▁▁▁▁▁▁▁▁▁▁▁▁▁▁▁▁▁▁
   // Scenario ④, alarm reset level reached for more than the off-delay duration
   // 
   // At point ④ on the graph, the signal actual_Value again falls below the alarm reset level 
   // (SP_ALM_H_VAL − SP_ALM_H_HYST_VAL).
   // 
   // Again, at this point, the off-delay timer starts; in the case of point ④, the signal actual_Value 
   // remains below the reset threshold for the full duration of the TIME_ALM_H_OFF_DEL and 
   // consequently, the alarm deactivates (msg_Alm_H goes to a low state), this is indicated in the 
   // middle msg_Alm_H graph.
   // 
   // 
   // 
   // ▁▁▁▁▁▁▁▁▁▁▁▁▁▁▁▁▁▁▁▁▁▁▁▁▁▁▁▁▁▁▁▁▁▁▁▁▁▁▁▁▁▁▁▁
   // Scenario ⑤, alarm is disabled
   // 
   // If the alarm is disabled (CONFIG_ALM_H_ENABLE = 0) then the alarm will never activate 
   // (msg_Alm_H is always in a low state), this is indicated in the lower msg_Alm_H graph.
   // 
   // Note:    The timer for disabled alarms and warnings is permanently set to zero.
   // 
   // 
   // ▁▁▁▁▁▁▁▁▁▁▁▁▁▁▁▁▁▁▁▁▁▁▁▁▁▁▁▁▁▁▁▁▁▁▁▁▁▁▁▁▁▁▁▁
   // 3.2.2     Low alarms and warnings
   // 
   // Low alarms and warnings are very similar to the high alarms of § 3.2.1, they do however work
   // in the opposite sense (the inequalities are reversed), low alarms and warnings are activated
   // when the actual_Value falls below, or is equal to, the SP_ALM_L_VAL, and deactivates when it
   // rises above SP_ALM_L_VAL + SP_ALM_L_HYST_VAL.
   // 
   // On and off delays work in exactly the same way as those for the high alarm.
   // 
   // A worked example of the low alarm is given in the online documentation for this block:
   // 
   // select this block in the project tree and press:
   //      SHIFT + F1
   // 
   // 
   // 
   // 
   // ▁▁▁▁▁▁▁▁▁▁▁▁▁▁▁▁▁▁▁▁▁▁▁▁▁▁▁▁▁▁▁▁▁▁▁▁▁▁▁▁▁▁▁▁
   // 3.2.3     Masking alarms and warnings
   // 
   // There are conditions where it can become necessary to mask (supress) alarms and warnings, a 
   // typical example could be a flow meter that monitors the flow into a filter; under normal 
   // conditions the flow meter would generate a low alarm if the flow into the filter were below a 
   // certain setpoint (indicating that the filter is becoming blocked).
   // 
   // It would be normal practice to supress this alarm when the filter was being cleaned, under 
   // these circumstances there would be no flow into the filter, but this would be a normal operating 
   // condition for the filter; the flow meter should only be monitoring for a low alarm during normal 
   // operation, not when the filter is being cleaned.
   // 
   // This suppression of an alarm or warning is referred to as “masking”, and there is a mask bit for 
   // each alarm and warning:
   // 
   //  ――――――――――――――――――――――――――――――――――――――――――
   //  SIGNAL           FUNCTION           TYPE   DETAILS
   //  ――――――――――――――――――――――――――――――――――――――――――
   //  mode_Alm_H_MaskOn    Masks the high alarm     Bool    1 = alarm masked, 0 = normal
   //  mode_Alm_L_MaskOn    Masks the low alarm    Bool    1 = alarm masked, 0 = normal
   //  mode_Wrn_H_MaskOn    Masks the high warning    Bool    1 = warning masked, 0 = normal
   //  mode_Wrn_L_MaskOn     Masks the low warning      Bool    1 = warning masked, 0 = normal
   //  ――――――――――――――――――――――――――――――――――――――――――
   //  Alarm and warning mask signals
   // 
   //  
   // Any alarm or warning that is masked (the mode_Xxx_Y_MaskOn = 1), will deactivate instantly 
   // (there is no off-delay) and will not reactivate activate (the msg_Xxx_Y will be set to zero), the 
   // effect is the same as if the CONFIG_XXX_Y_ENABLE bit were turned off.
   // 
   // The difference between the mask and the ENABLE signals is that the enable signal is a 
   // configuration of the instrument (it determines which alarms and warnings are configured for the 
   // particular instrument) and does not change at run-time (it is stored in static data block).
   // 
   // The mask signal on the other hand can be changed at run-time (either by some aspect of the 
   // Controller program or by the operator). The mask signal is stored in a dynamic data block and 
   // can be freely modified.
   // 
   // Note:    If an alarm or warning is not enabled (CONFIG_XXX_Y_ENABLE = 0), then the mask bit 
   //      (mode_Xxx_Y_MaskOn) will not do anything (setting it will not enable the alarm), in 
   //      fact if the alarm or warning is not enabled, the mask bit will be permanently set to 
   //      zero.
   // 
   // Masking alarms and warnings is the correct way to disable an alarm as part of the process 
   // operation of the plant.
   // 
   // When an alarm or warning goes from a masked condition to an unmasked condition (returns to 
   // normal operation), the on-delay timer will be reset and any alarm or warning condition will 
   // have to go back through the on-delay process before the alarm or warning can reactivate, this is 
   // true even if the alarm were active before being masked.
   // 
   // 
   // 
   // 
   // ▁▁▁▁▁▁▁▁▁▁▁▁▁▁▁▁▁▁▁▁▁▁▁▁▁▁▁▁▁▁▁▁▁▁▁▁▁▁▁▁▁▁▁▁
   // 3.2.4     A note on dynamically enabling alarms
   // 
   // In normal operations, alarms are either enabled or disabled as part of the instrument 
   // configuration and this configuration will not change during run-time; the enable signal 
   // (CONFIG_XXX_Y_ENABLE) is after all in a static data block. 
   // 
   // However, it is possible that the static data block is being used as a recipe block and as such it 
   // could be overloaded at some point during run-time.
   // 
   // Should the block detect a change in any of the CONFIG_XXX_Y_ENABLE; specifically, a rising 
   // edge, the block provided error checking to ensure that the associated alarm/warning timer 
   // (actual_Xxx_Y_Timer) is preset to correct TIME_XXX_Y_ON_DEL, this prevents the alarm/warning 
   // from activating instantly, if the actual_Value is outside the alarm/warning setpoint. A condition 
   // that could arise because the timer is set to zero while ever the alarm/warning is disabled.
   // 
   // Note:    This is a minor technical point, but it is a necessary error trapping mechanism — the 
   //      situation could arise even if it is unlikely.
   // 
   // 
   // 
   // ▂▂▂▂▂▂▂▂▂▂▂▂▂▂▂▂▂▂▂▂▂▂▂▂▂▂▂▂▂▂▂▂▂▂▂▂▂▂▂▂▂▂▂▂
   // 3.3     Fault signals
   // 
   // There are four fault signals that can be produced by the block:
   // 
   // 
   //  ――――――――――――――――――――――――――――――――――――――――――
   //  SIGNAL           FUNCTION            TYPE   DETAILS
   //  ――――――――――――――――――――――――――――――――――――――――――
   //  msg_Flt_UnderRange   The instrument is more than   Bool    1 = under range, 0 = healthy
   //                 a percentage below the its 
   //                 minimum value
   //  msg_Flt_OverRange     The instrument is more than   Bool    1 = over range, 0 = healthy
   //                 a percentage above its 
   //                 maximum value
   //  msg_Flt_OutOfRange   Common fault, either       Bool    1 = out of range, 0 = healthy
   //                 under or over range
   //  msg_Flt_External     The instrument itself is    Bool    1 = fault, 0 = healthy
   //                 indicating a fault 
   //                 (hardwired signal)
   //  ――――――――――――――――――――――――――――――――――――――――――
   //  Block fault signals 
   // 
   // 
   // 
   // ▁▁▁▁▁▁▁▁▁▁▁▁▁▁▁▁▁▁▁▁▁▁▁▁▁▁▁▁▁▁▁▁▁▁▁▁▁▁▁▁▁▁▁▁
   // 3.3.1     Over, under and out of range fault signals
   // 
   // If the signal from the instrument the RAW_ANALOG signal, is outside the RANGE_RAW_MIN to 
   // RANGE_RAW_MAX range (red dotted area of the graph, Figure 3.1), the scaled instrument reading 
   // (actual_Value) will still be calculated correctly; however, an appropriate, over-range or 
   // under-range (msg_Flt_OverRange or msg_Flt_UnderRange) signal will be generated to indicate 
   // that the instrument signal is outside of its calibrated range and is potentially no longer accurate.
   // 
   // Some tolerance is permitted before either the msg_Flt_OverRange or msg_Flt_UnderRange 
   // signals is activated (this is to prevent nuisance alarms — most instruments are tolerant of slight 
   // over and under shoot readings). 
   // 
   // The tolerance applied to the out of range signals is a percentage of the raw range of the 
   // instrument (the raw range being RANGE_RAW_MAX − RANGE_RAW_MIN). 
   // 
   // The tolerance to be applied is given in the parameter RANGE_OOR_PERCENT, this is a real 
   // (floating point) number in the range 0.0-10.0%.
   // 
   // If the tolerance for the instrument is not known, a generic value of 2.5% should be used.
   // 
   // The out of range tolerance absolute value (in terms of the RAW_ANALOG rather than as a 
   // percentage) is calculated as:
   // 
   // 
   // 
   // ┌─────────────────────────────────────┐
   // │                            (RANGE_RAW_MAX ─ RANGE_RAW_MIN) ╳ RANGE_OOR_PERCENT  │
   // │ calcRawOOR =  ―――――――――――――――――――――――――――― │
   // │                      100              │
   // └─────────────────────────────────────┘
   // 
   // Thus, if RANGE_RAW_MIN is 0, RANGE_RAW_MAX is 27648 and a RANGE_OOR_PERCENT of 2.5% is 
   // selected, the absolute out of range value (calcRawOOR in the above equation) has a calculated
   //  value of 691. 
   // 
   // In this example, the msg_Flt_OverRange signal would activate when RAW_ANALOG 
   // exceeded a value of RANGE_RAW_MAX + 691 (or 28,339). The msg_Flt_UnderRange signal would 
   // activate when RAW_ANALOG fell below a value of RANGE_RAW_MIN − 691 (or −691).
   // 
   // The RANGE_OOR_PERCENT is applied directly to the RAW_ANALOG signal, however, because the 
   // instrument is considered to be linear, the same calculation can also be ap-plied directly to the 
   // scaled reading of the instrument (actual_Value). 
   // 
   // In the example given in § 2.1, the instrument spans the range of -100 l/s to +100 l/s 
   // (i.e. RANGE_SCALE_MIN = -100 and RANGE_SCALE_MAX = +100) then the scaled range of the 
   // instrument is 200 l/s (RANGE_SCALE_MAX − RANGE_SCALE_MIN) and the absolute out of range 
   // value would be 2.5% of the scaled range (or 5 l/s). thus, the msg_Flt_OverRange signal would 
   // activate above 105 l/s and the msg_Flt_UnderRange signal would activate below −105 l/s.
   // 
   // Note:    If the range information supplied to the module is incorrect, either:
   //        •   RAW_MAX <= RAW_MIN or
   //        •   SCALE_MAX <= SCALE_MIN
   //      Then all the out of range signals are activated
   // 
   // 
   // 
   // ▁▁▁▁▁▁▁▁▁▁▁▁▁▁▁▁▁▁▁▁▁▁▁▁▁▁▁▁▁▁▁▁▁▁▁▁▁▁▁▁▁▁▁▁
   // Common out of range signal
   // 
   // There is a third out of range signal: msg_Flt_OutOfRange, this signal is a common signal that 
   // just indicates the instrument is out of its calibrated range (it does not specify whether it is over 
   // or under range). It is activated if either the msg_Flt_OverRange or msg_Flt_UnderRange signal is 
   // active.
   // 
   // 
   // 
   // ▁▁▁▁▁▁▁▁▁▁▁▁▁▁▁▁▁▁▁▁▁▁▁▁▁▁▁▁▁▁▁▁▁▁▁▁▁▁▁▁▁▁▁▁
   // 3.3.2     External fault signal
   // 
   // The external fault is an optional hardwired signal from the instrument, it indicates that the 
   // instrument itself is registering that there is some problem. Such external fault signals are more 
   // commonly associated with complex instruments (mass flow metres, ultrasonic level 
   // transducers, analytical instruments &c.) rather than the more simplistic instruments (pressure 
   // sensors, temperature transmitters &c.).
   // 
   // Typical examples of external faults would be:
   // 
   //    •   No medium present in a mass flow meter (if the instrument were measuring liquid 
   //      flow and the pipe had become empty)
   // 
   //    •   Foam indication from an ultrasonic level transducer (preventing an accurate level 
   //      reading)
   // 
   // Such fault signals are generally indicated via a hardwired digital input to the Controller.
   // 
   // The external fault signal (if used) is passed to the block as the parameter: EXT_FAULT
   // 
   //  ――――――――――――――――――――――――――――――――――――――――――
   //  PARAMETER          FUNCTION            TYPE   DETAILS
   //  ――――――――――――――――――――――――――――――――――――――――――
   //  EXT_FAULT        Hardwired signal indicating    Bool    1 = fault, 0 = healthy
   //                 the instrument is in a fault 
   //                 condition
   //  ――――――――――――――――――――――――――――――――――――――――――
   //  Block external fault parameter 
   // 
   // If the EXT_FAULT signal is not required, the input should be set to _false.
   // 
   // If the instrument generates a fault signal in the opposite sense, i.e. 0 = fault and 1 = healthy (this 
   // is a common fail-safe condition, that generates a fault signal if the instrument is disconnected 
   // or a wire break occurs), then a normally closed contact should be applied to the EXT_FAULT 
   // parameter to invert the signal into the block (see Figure 3.4):
   // 
   // 
   //                       ┌─────────────
   //    ───────────────────┤ FC02001 
   //                       ├───────────────┤
   //                           "FC001" ─┤ RAW_ANALOG           │
   //                       │               │
   //         "FC001_FAULT"           │               │
   //      ────┤╱├──────────┤ EXT_FAULT                │
   //                       │               │
   //                       │               │
   //   "DB02001_St_StdInstAnalogRead".FC001 ─┤ STATIC_DATA             │
   //                       │
   //   "DB22001_Dy_StdInstAnalogRead".FC001 ─┤ DYNAMIC_DATA
   //                       │
   //                       │
   // 
   // 
   // If the EXT_FAULT parameter is activated (set to 1), the corresponding fault signal within the 
   // dynamic data (msg_Flt_External) will be activated, there are no delays or other filtering 
   // associated with this signal.
   // 
   // Note:    The external fault does not in any way impact the reading and scaling of the 
   //      instrument or the production of any alarms or warnings.
   // 
   // 
   // 
   // ▂▂▂▂▂▂▂▂▂▂▂▂▂▂▂▂▂▂▂▂▂▂▂▂▂▂▂▂▂▂▂▂▂▂▂▂▂▂▂▂▂▂▂▂
   // 3.4     Operating mode
   // 
   // This block  supports various operating modes:
   // 
   //    •   Simulation mode
   //    •   Remote/local mode
   //    •   Faceplate disabled mode
   // 
   // Examining these in turn:
   // 
   // 
   // ▁▁▁▁▁▁▁▁▁▁▁▁▁▁▁▁▁▁▁▁▁▁▁▁▁▁▁▁▁▁▁▁▁▁▁▁▁▁▁▁▁▁▁▁
   // 3.4.1     Simulation mode
   // 
   // The instrument can be switched to a simulation mode, in which the actual reading from the 
   // instrument is replaced by a simulated value provided by the operator. 
   // 
   // Simulation mode is generally used during testing, but can also be applied in a process 
   // environment if a fault condition is detected within the instrument; this scenario allows the plant 
   // to continue operating (albeit under some degree of manual control) until the instrument is 
   // repaired or replaced.
   // 
   // The following data points are associated with the simulation mode:
   // 
   //  ――――――――――――――――――――――――――――――――――――――――――
   //  SIGNAL           FUNCTION            TYPE   DETAILS
   //  ――――――――――――――――――――――――――――――――――――――――――
   //  CONFIG_SIM_DISABLE      Prevents simulation mode   Bool    1 = no sim, 0 = sim permitted
   //                 being activated under all 
   //                 circumstances
   // 
   //  mode_SimOn        Activates simulation mode,    Bool    1 = sim on, 0 = sim off
   //                 if active, the scaled reading 
   //                 of the instrument (Value) will 
   //                 be set to mode_SimValue
   // 
   //  mode_SimValue      Scaled instrument reading   Real    Simulated instrument value
   //                 (Value) will be set to this if 
   //                 simulation mode is on
   //                 (CONFIG_SIM_OFF = 0 and 
   //                 mode_SimOn = 1)
   // 
   //  status_SimOn       Status indication, shows if    Bool    1 = sim active, 0 = Sim off
   //                 simulation mode is active
   //  ――――――――――――――――――――――――――――――――――――――――――
   // 
   // 
   // Simulation mode can only be activated by the operator via a faceplate available at the 
   // supervisory system (SCADA/HMI).
   // 
   // If simulation mode is disabled (configuration signal CONFIG_SIM_OFF is set to 1), then the 
   // simulation mode cannot be turned on under any circumstances, the option is greyed out on the 
   // supervisory system faceplate and the block will constantly reset the mode_SimOn signal.
   // 
   // If simulation mode is permitted (CONFIG_SIM_OFF = 0), then setting mode_SimOn to 1 will 
   // activate simulation mode and the scaled instrument value (actual_Value) will be set to the 
   // value stored in mode_SimValue:
   // 
   //           i.e. actual_Value = mode_SimValue
   // 
   // and all fault messages will be reset.
   // 
   // The operator can set and adjust the simulation value (mode_SimValue) from the instrument
   // faceplate on the supervisory system. The simulation value can be adjusted at any time by the 
   // operator (even if simulation mode has not been activated), but will not be applied until 
   // simulation mode is turned on (mode_SimOn = 1). 
   // 
   // If simulation mode is completely disabled (CONFIG_SIM_OFF is set to 1) then the operator will
   // not be able to adjust the simulated value (mode_SimValue will be greyed out on the faceplate).
   // 
   // 
   // 
   // ▁▁▁▁▁▁▁▁▁▁▁▁▁▁▁▁▁▁▁▁▁▁▁▁▁▁▁▁▁▁▁▁▁▁▁▁▁▁▁▁▁▁▁▁
   // 3.4.2     Remote/local mode
   // 
   // Remote and local operating modes refer to the supervisory system that has control of the 
   // instrument (i.e. which system can write to the device and change the operating mode of the 
   // device). 
   // 
   // This type of mode is usual present where a plant has a remote central control location (a control 
   // room) that normally controls the device (remote control), but also has a field panel with a local 
   // HMI that an operator in the field can select to take over control of the device (local control) for 
   // maintenance purposes.
   // 
   // The modes are as follows (and are mutually exclusive, only one will be active):
   // 
   //    Remote        Only the remote system in the control room can 
   //                 control the device
   // 
   //    Local            A local system has taken control of the device and the remote 
   //                 system can no longer issue commands to it
   // 
   //    Remote/local disabled   The system does not use remote/local modes and any 
   //      (ALL mode)     supervisory system can issue commands to the device 
   //  
   // Remote/local control is generally handled by the supervisory systems themselves; however, the 
   // supervisory systems need a storage area per device to record which mode that device is in, local 
   // control is often activated by a panel key-switch, that changes the state of several devices from 
   // remote to local (usually all the devices controlled by the local panel).
   // 
   // The block simply identifies the remote/local mode from the mode signals and configuration 
   // signals provided to the block.
   // 
   // For systems that do not use remote/local modes (any supervisory system can control the device, 
   // or control is determined by operator privileges), the remote/local modes can be disabled 
   // (CONFIG_RL_ENABLE is set to zero) and the device is effectively in ALL mode (any system can 
   // control the device).
   // 
   // If remote/local operation is in use, the supervisory system that does not have control will still 
   // display all the information from the device, but will not be able to control the device (it could not 
   // for example, activate simulation mode) and all control function (faceplate functions) will be 
   // greyed out.
   // 
   // The following signals are associated with remote/local/all modes:
   // 
   // 
   //  ――――――――――――――――――――――――――――――――――――――――――
   //  SIGNAL           FUNCTION            TYPE   DETAILS
   //  ――――――――――――――――――――――――――――――――――――――――――
   //  CONFIG_RL_ENABLE   Allows Remote and Local      Bool    1 = Remote/local selected
   //                 modes to be selected        0 = All mode is active
   // 
   //  mode_RemoteOn       Activates remote mode     Bool    1 = remote mode on, 
   //                 CONFIG_RL_ENABLE must = 1    0 = remote mode off
   // 
   //  mode_LocalOn     Activates local mode          Bool    1 = local mode on, 
   //                 CONFIG_RL_ENABLE must = 1    0 = remote mode off
   // 
   //  status_RemoteOn      Status remote mode on     Bool    1 = remote mode on, 
   //                               0 = remote mode off
   // 
   //  status_LocalOn       Status local mode on      Bool 1 = local mode on, 
   //                               0 = local mode off
   // 
   //  status_RLOff       Status ALL mode is on = 0    Bool 1 = ALL mode on, 
   //                               0 = ALL mode off
   //  ――――――――――――――――――――――――――――――――――――――――――
   //  Block remote/local signals 
   // 
   // By default, remote/local is disabled — ALL mode is selected (CONFIG_RL_ENABLE = 0).
   // 
   // 
   // 
   // 
   // ▁▁▁▁▁▁▁▁▁▁▁▁▁▁▁▁▁▁▁▁▁▁▁▁▁▁▁▁▁▁▁▁▁▁▁▁▁▁▁▁▁▁▁▁
   // 3.4.3     Faceplate disable mode
   // 
   // It is possible to disable the supervisory system faceplate from within the block, the con-figuration 
   // signal:
   // 
   // 
   //  ――――――――――――――――――――――――――――――――――――――――――
   //  SIGNAL           FUNCTION            TYPE   DETAILS
   //  ――――――――――――――――――――――――――――――――――――――――――
   //  CONFIG_FP_DISABLE     Disable the supervisory      Bool    1 = Faceplate disabled
   //                 system faceplate           0 = normal
   //  ――――――――――――――――――――――――――――――――――――――――――
   //  Block faceplate disable signal 
   // 
   // If the faceplate is disabled (CONFIG_FP_DISABLE = 1), the supervisory system will not allow the 
   // device faceplate to be opened (normally achieved by clicking the block icon or device symbol), 
   // this in turn prevents the operator from affecting the device in anyway, it would not, for example, 
   // be possible to put the device into simulation mode.
   // 
   // Similarly, if the faceplate is disabled, the module will set remote/local mode to ALL and will 
   // disable simulation mode.
   // 
   // 
   // 
   // ▂▂▂▂▂▂▂▂▂▂▂▂▂▂▂▂▂▂▂▂▂▂▂▂▂▂▂▂▂▂▂▂▂▂▂▂▂▂▂▂▂▂▂▂
   // 3.5     Block icon signals
   // 
   // This block has a partner block icon that represents the instrument and its various modes and 
   // status in a graphical format (block icon) that is displayed on a supervisory system (SCADA or HMI).
   // 
   // See the online documentation for this block — select the block in the project tree and press:
   //      SHIFT + F1
   // 
   // The supervisory system interface is available in section 3.7 of the online SMDS document.
   // 
   // 
   // 
   // ▁▁▁▁▁▁▁▁▁▁▁▁▁▁▁▁▁▁▁▁▁▁▁▁▁▁▁▁▁▁▁▁▁▁▁▁▁▁▁▁▁▁▁▁
   // 3.5.1     Understanding status signals
   // 
   // The status signals for faults, alarms and warnings are either duplicates of the message signals 
   // (signals beginning with msg_) or logical combinations of them.
   // 
   // The following is a full list of the status signals:
   // 
   //  ――――――――――――――――――――――――――――――――――――――――――
   //  SIGNAL           FUNCTION            TYPE   DETAILS
   //  ――――――――――――――――――――――――――――――――――――――――――
   //  status_Alm_H        Identical to: msg_Alm_H    Bool    1 = high alm active, 0 = no alm
   // 
   //  status_Alm_L         Identical to: msg_Alm_L       Bool    1 = low alm active, 0 = no alm
   // 
   //  status_Wrn_H        Identical to: msg_Wrn_H    Bool    1 = high wrn active, 0 = no wrn
   // 
   //  status_Wrn_L         Identical to: msg_Wrn_L     Bool    1 = low wrn active, 0 = no wrn
   // 
   //  status_Alm_H_Mask     High alarm is masked     Bool    1 = masked, 0 = normal
   // 
   //  status_Alm_L_Mask   Low alarm is masked      Bool    1 = masked, 0 = normal
   // 
   //  status_Wrn_H_Mask      High warning is masked    Bool    1 = masked, 0 = normal
   // 
   //  status_Wrn_L_Mask       Low warning is masked     Bool    1 = masked, 0 = normal
   // 
   //  status_Alm_H_Dis         High alarm is disabled       Bool    1 = disabled, 0 = normal
   // 
   //  status_Alm_L_Dis       Low alarm is disabled        Bool    1 = disabled, 0 = normal
   // 
   //  status_Wrn_H_Dis          High warning is disabled      Bool    1 = disabled, 0 = normal
   // 
   //  status_Wrn_L_Dis           Low warning is disabled       Bool    1 = disabled, 0 = normal
   // 
   //  status_Fault       Indicates any of the msg_Flt    Bool    1 = fault active, 0 = healthy
   //                 signals are active:
   //                  msg_Flt_UnderRange
   //                  msg_Flt_OverRange
   //                  msg_Flt_OutOfRange
   //                  msg_Flt_External 
   // 
   //  status_SimOn       Status simulation mode on     Bool    1 = sim on, 0 = sim off
   // 
   //  status_RemoteOn      Status remote mode on     Bool    1 = rem on, 0 = rem off
   // 
   //  status_LocalOn       Status local mode on      Bool    1 = loc on, 0 = loc off 
   // 
   //  status_RLOff       Status ALL mode is on           Bool    1 = ALL mode on, 
   //                               0 = ALL mode off
   //  ――――――――――――――――――――――――――――――――――――――――――
   //  Block status signals 
   // 
   // 
   // 
   // ▁▁▁▁▁▁▁▁▁▁▁▁▁▁▁▁▁▁▁▁▁▁▁▁▁▁▁▁▁▁▁▁▁▁▁▁▁▁▁▁▁▁▁▁
   // 3.5.2     String constants for tag name and units
   // 
   // The STATIC_DATA structure holds two string values:
   // 
   //  UT02001_St_InstAnalogRead (full contents)
   //  ――――――――――――――――――――――――――――――――――――――――――
   //  SIGNAL NAME          FUNCTION                     TYPE
   //  ――――――――――――――――――――――――――――――――――――――――――
   //  INFO_TAG          INFORMATION — Instrument ID tag          String[20]
   // 
   //  INFO_UNITS          INFORMATION — Engineering units of the instrument  String[10]
   //                        (unit of measure)
   //  ――――――――――――――――――――――――――――――――――――――――――
   //  String constants for the instrument
   // 
   // These two strings allow the supervisory system to populate the instrument tag (e.g. FIC001) and 
   // the engineering units applicable to the instrument (L/s for example) directly from the data 
   // stored in the PLC; it means the block icon can be used directly within the supervisory system 
   // graphic without customisation; all the data will be populated directly at runtime.
   // 
   //                ━━━   ⬙⬙⬙⬙⬙⬙   ━━━
END_REGION

REGION Network 3: Block description — Sections 4 to 11
   // ▄▄▄▄▄▄▄▄▄▄▄▄▄▄▄▄▄▄▄▄▄▄▄▄▄▄▄▄▄▄▄▄▄▄▄▄▄▄▄▄▄▄▄▄
   // 4.     PARAMETERS
   // 
   // 
   // The following parameters are associated with the block:
   // 
   //  
   //  ――――――――――――――――――――――――――――――――――――――――――
   //  PARAM         FUNCTION                    TYPE      IN-OUT 
   //  ――――――――――――――――――――――――――――――――――――――――――
   //  SYS_SIGNALS      Common system signals              UT21000    In
   //           logic and timing signals for parametric access
   // 
   //  RAW_ANALOG      The unscaled analogue input (input word         Word     In
   //           address for the IO card to which the instrument 
   //           is connected)
   // 
   //  EXT_FAULT     Optional external fault signal for the instrument      Bool      In
   //           (1 = fault, 0 = healthy). If not required, set 
   //           permanently to _False
   // 
   //  STATIC_DATA     Data structure that holds the configuration data     UT02001    In
   //           for the instrument (raw range, scaled range 
   //           alarm and warning values, filtering times, 
   //           hysteresis values &c.)
   // 
   //  DYNAMIC_DATA      Data structure that holds the live data for the       UT22001    InOut
   //           instrument (its reading in engineering units, 
   //           any alarms or warnings that may be active, 
   //           current timer values, selected operating 
   //           mode &c.)
   //  ――――――――――――――――――――――――――――――――――――――――――
   // 
   //                ━━━   ⬙⬙⬙⬙⬙⬙   ━━━
   // 
   // 
   // 
   // ▄▄▄▄▄▄▄▄▄▄▄▄▄▄▄▄▄▄▄▄▄▄▄▄▄▄▄▄▄▄▄▄▄▄▄▄▄▄▄▄▄▄▄▄
   // 5.     DATA STRUCTURES AND USAGE (AND INSTANCE DATA BLOCKS)
   // 
   // 
   // The block has the following associated data structure:
   // 
   // 
   //  ――――――――――――――――――――――――――――――――――――――――――
   //  DATA STRUCTURE             DESCRIPTION
   //  ――――――――――――――――――――――――――――――――――――――――――
   //  UT01000_St_SysRevision          Revision information for this block    See FC01001
   //  UT01001_St_SysLicence           Licence information for this block  See FC01001
   //  UT21000_Dy_SysSignals           System signals for logic and timing  See FC01001
   // 
   //  UT02001_St_InstAnalogRead      Static data structure for an analogue instrument.
   //                     Holds configuration information, instrument ranges 
   //                     and scaling, alarm/warning thresholds &c.
   // 
   //  UT22001_Dy_InstAnalogRead        Dynamic data structure for an analogue instrument.
   //                     Current scaled instrument reading, alarm status, 
   //                     operating modes, timer values &c.
   //  ――――――――――――――――――――――――――――――――――――――――――
   // 
   // 
   // 
   // ▂▂▂▂▂▂▂▂▂▂▂▂▂▂▂▂▂▂▂▂▂▂▂▂▂▂▂▂▂▂▂▂▂▂▂▂▂▂▂▂▂▂▂▂
   // 5.1     UT02001_St_InstAnalogRead
   // 
   // The static data structure for an analogue instrument.
   // 
   // 
   //  UT02001_St_InstAnalogRead (full contents)
   //  ――――――――――――――――――――――――――――――――――――――――――
   //  SIGNAL NAME          FUNCTION                     TYPE
   //  ――――――――――――――――――――――――――――――――――――――――――
   //  CONFIG_ALM_H_ENABLE  CONFIG — High alarm is enabled          Bool
   //                      (1 = enabled, 0 = no alarm) 
   //  CONFIG_ALM_L_ENABLE   CONFIG — Low alarm is enabled           Bool
   //                      (1 = enabled, 0 = no alarm)
   //  CONFIG_WRN_H_ENABLE     CONFIG — High warning is enabled         Bool
   //                      (1 = enabled, 0 = no warning)
   //  CONFIG_WRN_L_ENABLE     CONFIG — Low warning is enabled          Bool
   //                      (1 = enabled, 0 = no warning)
   //  CONFIG_FP_DISABLE      CONFIG — Faceplate is disabled           Bool
   //                      (1 = no Faceplate, 0 = normal)
   //  CONFIG_SIM_DISABLE    CONFIG — Simulation is disabled            Bool
   //                      (1 = no Simulation, 0 = normal)
   //  CONFIG_RL_ENABLE    CONFIG — Remote/local mode enabled       Bool
   //                      (1 = enabled, 0 = all mode)
   // 
   //  RANGE_RAW_MIN       RANGE — Minimum value of the raw analogue    Int
   //                     signal (at the card)
   //  RANGE_RAW_MAX      RANGE — Maximum value of the raw analogue      Int
   //                     signal (at the card)
   //  RANGE_SCALE_MIN      RANGE — Minimum value of the scaled analogue     Real
   //                     signal [engineering units]
   //  RANGE_SCALE_MAX     RANGE — Maximum value of the scaled analogue    Real
   //                     signal [engineering units]
   //  RANGE_OOR_PERCENT      RANGE — Out of range percentage, beyond which    Real
   //                     the instrument is out of range
   // 
   //  INFO_TAG          INFORMATION — Instrument ID tag          String[20]
   // 
   //  INFO_UNITS          INFORMATION — Engineering units of the instrument  String[10]
   //                        (unit of measure)
   // 
   //  SP_ALM_H_VAL       SETPOINT — High alarm threshold value         Real
   //                      [engineering units]
   //  SP_ALM_L_VAL       SETPOINT — Low alarm threshold value       Real
   //                      [engineering units]
   //  SP_WRN_H_VAL         SETPOINT — High warning threshold value        Real
   //                      [engineering units]
   //  SP_WRN_L_VAL       SETPOINT — Low warning threshold value      Real
   //                      [engineering units]
   //  SP_ALM_H_HYST_VAL     SETPOINT — High alarm hysteresis value        Real
   //                      [engineering units]
   //  SP_ALM_L_HYST_VAL     SETPOINT — Low alarm hysteresis value         Real
   //                      [engineering units]
   //  SP_WRN_H_HYST_VAL    SETPOINT — High warning hysteresis value       Real
   //                      [engineering units]
   //  SP_WRN_L_HYST_VAL     SETPOINT — Low warning hysteresis value        Real
   //                      [engineering units]
   // 
   //  TIME_ALM_H_ON_DEL    TIMER — High alarm on delay time          Real
   //                      (activation delay), [seconds]
   //  TIME_ALM_L_ON_DEL     TIMER — Low alarm on delay time           Real
   //                      (activation delay), [seconds]
   //  TIME_WRN_H_ON_DEL       TIMER — High warning on delay time         Real
   //                      (activation delay), [seconds]
   //  TIME_WRN_L_ON_DEL        TIMER — Low warning on delay time          Real
   //                      (activation delay), [seconds]
   //  TIME_ALM_H_OFF_DEL      TIMER — High alarm off delay time           Real
   //                      (deactivation delay), [seconds]
   //  TIME_ALM_L_OFF_DEL       TIMER — Low alarm off delay time            Real
   //                      (deactivation delay), [seconds]
   //  TIME_WRN_H_OFF_DEL      TIMER — High warning off delay time          Real
   //                      (deactivation delay), [seconds]
   //  TIME_WRN_L_OFF_DEL      TIMER — Low warning off delay time           Real
   //                      (deactivation delay), [seconds]
   //  ――――――――――――――――――――――――――――――――――――――――――
   // 
   // 
   // 
   // ▂▂▂▂▂▂▂▂▂▂▂▂▂▂▂▂▂▂▂▂▂▂▂▂▂▂▂▂▂▂▂▂▂▂▂▂▂▂▂▂▂▂▂▂
   // 5.2      UT22001_Dy_InstAnalogRead
   // 
   // The static data structure for an analogue instrument.
   // 
   // 
   // 
   //  UT22001_Dy_InstAnalogReadl (full contents)
   //  ――――――――――――――――――――――――――――――――――――――――――
   //  SIGNAL NAME          FUNCTION                     TYPE
   //  ――――――――――――――――――――――――――――――――――――――――――
   //  status_ConfigError       STATUS — Raw or scaled range configuration error   Bool
   //                      (1 = Config error, 0 = OK)
   //  status_Alm_H         STATUS — High alarm is active           Bool
   //                      (1 = alarm active, 0 = no alarm)
   //  status_Alm_L          STATUS — Low alarm is active            Bool
   //                      (1 = alarm active, 0 = no alarm)
   //  status_Wrn_H         STATUS — High warning is active          Bool
   //                      (1 = warning active, 0 = no warning)
   //  status_Wrn_L          STATUS — Low warning is active           Bool
   //                      (1 = warning active, 0 = no warning)
   //  status_Alm_H_Mask       STATUS — High alarm is masked             Bool
   //                      (1 = alarm masked, 0 = normal)
   //  status_Alm_L_Mask        STATUS — Low alarm is masked              Bool
   //                      (1 = alarm masked, 0 = normal)
   //  status_Wrn_H_Mask       STATUS — High warning is masked            Bool
   //                      (1 = warning masked, 0 = normal)
   //  status_Wrn_L_Mask        STATUS — Low warning is masked             Bool
   //                      (1 = warning masked, 0 = normal)
   //  status_Alm_H_Dis           STATUS — High alarm is disabled            Bool
   //                      (1 = alarm disabled, 0 = normal)
   //  status_Alm_L_Dis            STATUS — Low alarm is disabled             Bool
   //                      (1 = alarm disabled, 0 = normal)
   //  status_Wrn_H_Dis           STATUS — High warning is disabled           Bool
   //                      (1 = warning disabled, 0 = normal)
   //  status_Wrn_L_Dis            STATUS — Low warning is disabled            Bool
   //                      (1 = warning disabled, 0 = normal)
   //  status_Fault            STATUS — Instrument is in fault             Bool
   //                      (1 = fault present, 0 = healthy)
   //  status_SimOn           STATUS — Instrument is in simulation mode     Bool
   //                      (1 = Simulation mode, 0 = normal)
   //  status_RemoteOn       STATUS — Instrument is in remote mode        Bool
   //                      (1 = Remote mode, 0 = normal)
   //  status_LocalOn         STATUS — Instrument is in local mode          Bool
   //                      (1 = Local mode, 0 = normal)
   //  status_RLOff         STATUS — Instrument is in ALL mode         Bool
   //                      (1 = ALL mode, 0 = normal)
   // 
   //  mode_Alm_H_MaskOn     MODE — Masks the high alarm             Bool    
   //                    (1 = alarm masked, 0 = normal)
   //  mode_Alm_L_MaskOn     MODE — Masks the low alarm            Bool    
   //                    (1 = alarm masked, 0 = normal)
   //  mode_Wrn_H_MaskOn     MODE — Masks the high warning            Bool    
   //                    (1 = warning masked, 0 = normal)
   //  mode_Wrn_L_MaskOn      MODE — Masks the low warning                 Bool    
   //                    (1 = warning masked, 0 = normal)
   //  mode_SimOn         MODE — Simulation mode               Bool
   //                    (1 = sim mode active, 0 = normal)
   //  mode_SimValue       MODE — Simulation value               Real
   //                    (engineering units)
   //  mode_LocalOn         MODE — Local HMI control enabled           Bool
   //                    (1 = active, 0 = disabled or N/A)
   //  mode_RemoteOn        MODE — Remote SCADA control enabled       Bool
   //                    (1 = active, 0 = disabled or N/A)
   // 
   //  msg_Alm_H         MESSAGE — Alarm - high alarm is active        Bool
   //  msg_Alm_L          MESSAGE — Alarm - low alarm is active          Bool
   //  msg_Wrn_H          MESSAGE — Warning - high warning is active      Bool
   //  msg_Wrn_L          MESSAGE — Warning - low warning is active        Bool
   //  msg_Flt_External         MESSAGE — Fault - external fault signal is active      Bool
   //  msg_Flt_OverRange¹     MESSAGE — Fault - instrument is over-range       Bool
   //  msg_Flt_UnderRange¹      MESSAGE — Fault - instrument is under-range       Bool
   //  msg_Flt_OutOfRange¹      MESSAGE — Fault - instrument is out-of-range        Bool
   // 
   //  batch_ID         BATCH — Booking ID (optional for batch operations)   Int
   // 
   //  actual_Value          ACTUAL — SCALED INSTRUMENT VALUE         Real
   //                      [engineering units]
   //  actual_Alm_H_Timer      ACTUAL — Timer value — alarm high operation     Real
   //                      timer [seconds]
   //  actual_Alm_L_Timer       ACTUAL — Timer value — alarm low operation    Real
   //                      timer [seconds]
   //  actual_Wrn_H_Timer      ACTUAL — Timer value — warning high operation    Real
   //                      timer [seconds]
   //  actual_Wrn_L_Timer       ACTUAL — Timer value — warning low operation      Real
   //                      timer [seconds]
   // 
   //  $pret_AlmHEn           INTERNAL — Edge retention (+ve) alarm high en      Bool
   //  $Pret_AlmLEn            INTERNAL — Edge retention (+ve) alarm low en     Bool
   //  $pret_WrnHEn           INTERNAL — Edge retention (+ve) warning high en     Bool
   //  $pret_WrnLEn            INTERNAL — Edge retention (+ve) warning low en       Bool
   //  ――――――――――――――――――――――――――――――――――――――――――
   //  ¹        msg_Flt_OverRange, msg_Flt_UnderRange and msg_Flt_OutOfRange will all
   //      activate if a configuration error is active status_ConfigError = 1, actual_Value will 
   //      also be set to zero under these conditions.
   // 
   // With the exception of the flowing, all these signals are discussed in the previous sections, the 
   // outstanding items are firstly:
   // 
   //      batch_ID
   // 
   // The batch_ID is not required for normal use; it is only used where a “booking” system is used 
   // (common in batch and routing applications). Such booking applications can acquire the device 
   // if it is free and reserve it for a particular phase of the batch. Batch applications are a topic in 
   // their own right and are discussed separately in the online User Guide.
   // 
   // Next:
   //      actual_Alm_H_Timer	Real
   //      actual_Alm_L_Timer	Real
   //      actual_Wrn_H_Timer	Real
   //      actual_Wrn_L_Timer	Real
   // 
   // These data points hold the actual value of the running timer for each of the alarms/warnings, 
   // both on and off-delay timers used the same timer within the block (the timers are mutually 
   // exclusive, only one will be running at once for each alarm or warning — hence only one timer is
   // needed for each alarm or warning).
   // 
   // Each timer counts down from the TIME_ values (UT02001_St_InstAnalogRead) to zero in 200 ms
   // intervals.
   // 
   // Finally:
   //      $pret_AlmHEn
   //      $Pret_AlmLEn
   //      $pret_WrnHEn
   //      $pret_WrnLEn
   // 
   // These are internal working signals (all signals the start with a $ are internal working signals 
   // used by the block). In this instance they are used to detect a rising edge on each of the alarm 
   // and warning enable signals. 
   // 
   //                ━━━   ⬙⬙⬙⬙⬙⬙   ━━━
   // 
   // 
   // 
   // ▄▄▄▄▄▄▄▄▄▄▄▄▄▄▄▄▄▄▄▄▄▄▄▄▄▄▄▄▄▄▄▄▄▄▄▄▄▄▄▄▄▄▄▄
   // 6.     CONSTANTS AND TEMPORARY (LOCAL) DATA
   // 
   // 
   // The following constants and temporary data storage are used:
   // 
   // 
   //  Temporary (local) data
   //  ――――――――――――――――――――――――――――――――――――――――――
   //  SIGNAL NAME          FUNCTION                  TYPE
   //  ――――――――――――――――――――――――――――――――――――――――――
   //  revInfo             Revision information for the block         UT01000
   //  licInfo           Licensing information for the block      UT01001
   //  wrkAlmHEn          Working Alm_H is enabled and not masked   Bool
   //  wrkAlmLEn        Working Alm_L is enabled and not masked    Bool
   //  wrkWrnHEn           Working Wrn_H is enabled and not masked    Bool
   //  wrkWrnLEn           Working Wrn_L is enabled and not masked    Bool
   //  calcPart1           Scale value part 1 (RAW_ANALOG − RAW_MIN)   Real
   //  calcPart2           Scale value part 2 (SCALE_MAX − SCALE_MIN)   Real
   //  calcPart3           Scale value part 3 (RAW_MAX − RAW_MIN)     Real
   //  calcRawOOR        Calculated OOR absolute value          Real
   //  calcOverRange       Calculated over range limit (in raw units)    Real
   //  calcUnderRange       Calculated under range limit (in raw units)     Real
   //  calcHystAbs         Absolute hysteresis value           Real
   //  wrkHyst           Working hysteresis value            Real
   //  wrkOORPercent         Working out of range percentage          Real
   //  wrkInt           Working storage area (integer)          Int
   //  wrkReal           Working storage (Real)             Real
   //  wrkDInt           Working storage area (double integer)         DInt
   //  ――――――――――――――――――――――――――――――――――――――――――
   // 
   //                ━━━   ⬙⬙⬙⬙⬙⬙   ━━━
   // 
   // 
   // 
   // ▄▄▄▄▄▄▄▄▄▄▄▄▄▄▄▄▄▄▄▄▄▄▄▄▄▄▄▄▄▄▄▄▄▄▄▄▄▄▄▄▄▄▄▄
   // 7.     BLOCK CALLS
   // 
   // There are no PAL block calls from within this block.
   // 
   //                ━━━   ⬙⬙⬙⬙⬙⬙   ━━━
   // 
   // 
   // 
   // ▄▄▄▄▄▄▄▄▄▄▄▄▄▄▄▄▄▄▄▄▄▄▄▄▄▄▄▄▄▄▄▄▄▄▄▄▄▄▄▄▄▄▄▄
   // 8.     ASSOCIATED BLOCKS
   // 
   // 
   // This is a stand-alone block and is not associated with any other blocks.
   // 
   //                ━━━   ⬙⬙⬙⬙⬙⬙   ━━━
   // 
   // 
   // 
   // ▄▄▄▄▄▄▄▄▄▄▄▄▄▄▄▄▄▄▄▄▄▄▄▄▄▄▄▄▄▄▄▄▄▄▄▄▄▄▄▄▄▄▄▄
   // 9.     SYSTEM BLOCK CALLS AND SYSTEM DATA TYPES
   // 
   // There are no system block calls.
   // 
   //                ━━━   ⬙⬙⬙⬙⬙⬙   ━━━
   // 
   // 
   // 
   // ▄▄▄▄▄▄▄▄▄▄▄▄▄▄▄▄▄▄▄▄▄▄▄▄▄▄▄▄▄▄▄▄▄▄▄▄▄▄▄▄▄▄▄▄
   // 10.     SPECIAL PROPERTIES AND REQUIREMENTS
   // 
   // 
   // 
   // ▂▂▂▂▂▂▂▂▂▂▂▂▂▂▂▂▂▂▂▂▂▂▂▂▂▂▂▂▂▂▂▂▂▂▂▂▂▂▂▂▂▂▂▂
   // 10.1   Block optimisation
   // 
   // 
   // Block optimisation is ACTIVE for this block
   // 
   // 
   // 
   // ▂▂▂▂▂▂▂▂▂▂▂▂▂▂▂▂▂▂▂▂▂▂▂▂▂▂▂▂▂▂▂▂▂▂▂▂▂▂▂▂▂▂▂▂
   // 10.2   Calling requirements
   // 
   // 
   // There are no special calling requirements for this block.
   // 
   //                ━━━   ⬙⬙⬙⬙⬙⬙   ━━━
   // 
   // 
   // 
   // ▄▄▄▄▄▄▄▄▄▄▄▄▄▄▄▄▄▄▄▄▄▄▄▄▄▄▄▄▄▄▄▄▄▄▄▄▄▄▄▄▄▄▄▄
   // 11.     EXAMPLE USAGE
   // 
   // 
   // The following shows a typical deployment of FC02001:
   // 
   //                         ┌─────────────
   //      ───────────────────┤ FC02001 
   //                         ├───────────────┤
   //    "DB21001_DY_StdGlobalData".SysSignals ─┤ SYS_SIGNALS
   //                         │               │
   //                          "FC001" ─┤ RAW_ANALOG           │
   //                         │               │
   //           "FC001_FAULT"           │               │
   //        ────┤╱├──────────┤ EXT_FAULT                │
   //                         │               │
   //                         │               │
   //     "DB02001_St_StdInstAnalogRead".FC001 ─┤ STATIC_DATA             │
   //                         │
   //     "DB22001_Dy_StdInstAnalogRead".FC001 ─┤ DYNAMIC_DATA
   //                         │
   //                         │
   //                                         │
   //                                ─────────┘
   // 
   // 
   //               ━━━   ⬙⬙⬙⬙⬙⬙   ━━━
   // 
   // 
   // 
   // ██████████████ █ █ █ █  END   █ █ █ █ ██████████████
END_REGION

REGION Network 4: Current revision and modification history
   // ▄▄▄▄▄▄▄▄▄▄▄▄▄▄▄▄▄▄▄▄▄▄▄▄▄▄▄▄▄▄▄▄▄▄▄▄▄▄▄▄▄▄▄▄
   // MODIFICATION HISTORY
   // 
   // 
   // The revision data shown here, in the network comments, contains additional information 
   // reflecting the software development workflow under the version control system (VCS) employed 
   // to track all software changes.
   // 
   // The VCS in use is the Git Source Code Management system in conjunction with the GitHub online 
   // hosting system. The software in its entirety is available in the GitHub remote repository:
   // 
   //      https://github.com/practicalseries/PS2001-pal-software
   // 
   // The repository is public and can be freely copied (forked in GitHub terminology) and used 
   // under the MIT licence. 
   // 
   // The MIT licence is reproduced in full in the last network of this software module
   // 
   // 
   //  ―――――――――――――――――――――――――――――――――――――――――――
   //  DATE       REVISION            MASTER BRANCH      DEV
   //          (nnn.amm)   COMMIT TAG    (Base ---> Merge)    BRANCH   Author
   //  ———————————————————————————————————————————
   //  2021.02.18    001.000   D0002A-001.000   D0002 N/A     D0002B   M. Gledhill
   //                        FC02001 Migration to VCS — Released for test
   // 
   //  2021.02.18    000.801   D0002A-000.801   D0002 N/A     D0002B   M. Gledhill
   //                        FC02001 Migration to VCS — Released for test
   //  ———————————————————————————————————————————
   //   Where: nnn  =  Major revision
   //         a  =  Type (1-7 Development, 8 Proving, 9 Qualification, 0 Release)
   //       mm  =  Minor revision (must be 00 if a = 0)
   //         Block properties version number should be set to nn.a (only one decimal place)
   // 
   // ▄▄▄▄▄▄▄▄▄▄▄▄▄▄▄▄▄▄▄▄▄▄▄▄▄▄▄▄▄▄▄▄▄▄▄▄▄▄▄▄▄▄▄▄
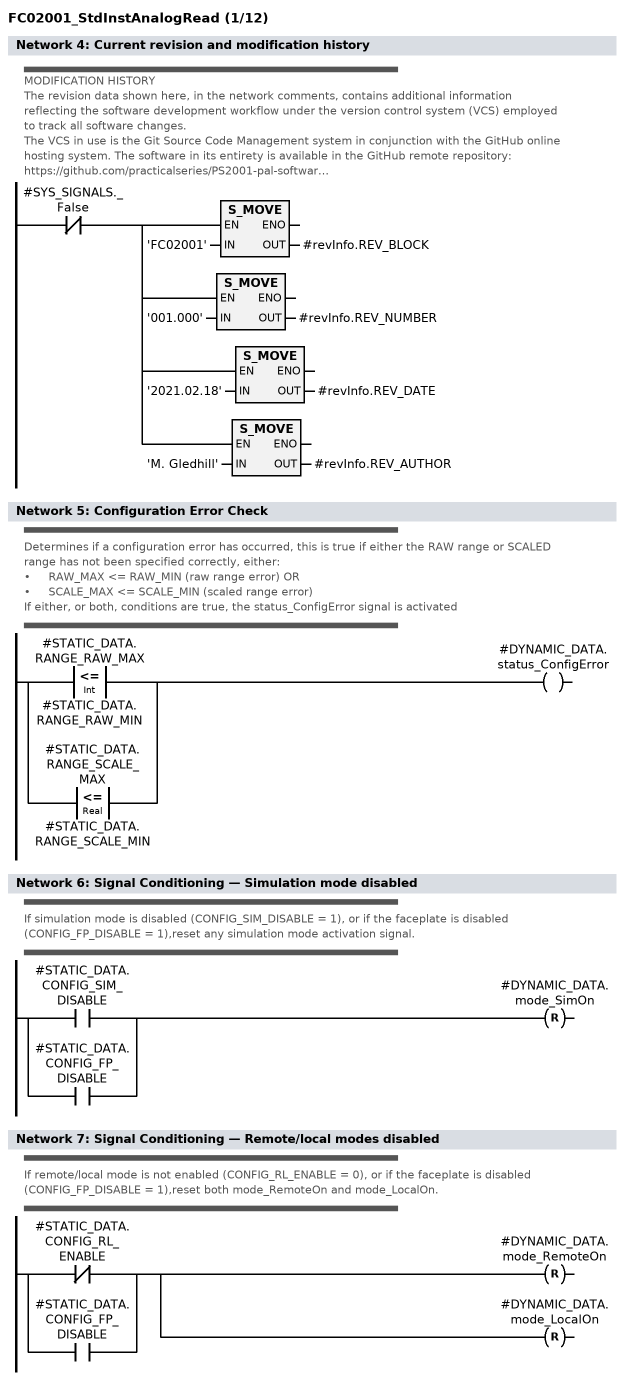
   RUNG wire#powerrail
      I_Contact( #SYS_SIGNALS._False )
      wire#w1
      S_Move(in := 'FC02001', out => #revInfo.REV_BLOCK)
   END_RUNG
   RUNG wire#w1
      S_Move(in := '001.000', out => #revInfo.REV_NUMBER)
   END_RUNG
   RUNG wire#w1
      S_Move(in := '2021.02.18', out => #revInfo.REV_DATE)
   END_RUNG
   RUNG wire#w1
      S_Move(in := 'M. Gledhill', out => #revInfo.REV_AUTHOR)
   END_RUNG
   // the same network as SCL:
   IF NOT #SYS_SIGNALS._False THEN
       #revInfo.REV_BLOCK := 'FC02001';
       #revInfo.REV_NUMBER := '001.000';
       #revInfo.REV_DATE := '2021.02.18';
       #revInfo.REV_AUTHOR := 'M. Gledhill';
   END_IF;
END_REGION

REGION Network 5: Configuration Error Check
   // ▀▀▀▀▀▀▀▀▀▀▀▀▀▀▀▀▀▀▀▀▀▀▀▀▀▀▀▀▀▀▀▀▀▀▀▀▀▀▀▀▀▀▀▀
   // 
   // Determines if a configuration error has occurred, this is true if either the RAW range or SCALED 
   // range has not been specified correctly, either:
   // 
   //    •   RAW_MAX <= RAW_MIN (raw range error) OR
   //    •   SCALE_MAX <= SCALE_MIN (scaled range error)
   // 
   // If either, or both, conditions are true, the status_ConfigError signal is activated
   // ▄▄▄▄▄▄▄▄▄▄▄▄▄▄▄▄▄▄▄▄▄▄▄▄▄▄▄▄▄▄▄▄▄▄▄▄▄▄▄▄▄▄▄▄
   RUNG wire#powerrail
      { S7_Templates := "SrcType := Int" } LE_Contact(in1 := #STATIC_DATA.RANGE_RAW_MAX, in2 := #STATIC_DATA.RANGE_RAW_MIN)
      wire#w1
      Coil( #DYNAMIC_DATA.status_ConfigError )
   END_RUNG
   RUNG wire#powerrail
      { S7_Templates := "SrcType := Real" } LE_Contact(in1 := #STATIC_DATA.RANGE_SCALE_MAX, in2 := #STATIC_DATA.RANGE_SCALE_MIN)
   END_RUNG wire#w1
   // the same network as SCL:
   #DYNAMIC_DATA.status_ConfigError := (#STATIC_DATA.RANGE_RAW_MAX <= #STATIC_DATA.RANGE_RAW_MIN) OR (#STATIC_DATA.RANGE_SCALE_MAX <= #STATIC_DATA.RANGE_SCALE_MIN);
END_REGION

REGION Network 6: Signal Conditioning — Simulation mode disabled
   // ▀▀▀▀▀▀▀▀▀▀▀▀▀▀▀▀▀▀▀▀▀▀▀▀▀▀▀▀▀▀▀▀▀▀▀▀▀▀▀▀▀▀▀▀
   // If simulation mode is disabled (CONFIG_SIM_DISABLE = 1), or if the faceplate is disabled 
   // (CONFIG_FP_DISABLE = 1),reset any simulation mode activation signal.
   // ▄▄▄▄▄▄▄▄▄▄▄▄▄▄▄▄▄▄▄▄▄▄▄▄▄▄▄▄▄▄▄▄▄▄▄▄▄▄▄▄▄▄▄▄
   RUNG wire#powerrail
      Contact( #STATIC_DATA.CONFIG_SIM_DISABLE )
      wire#w1
      R_Coil( #DYNAMIC_DATA.mode_SimOn )
   END_RUNG
   RUNG wire#powerrail
      Contact( #STATIC_DATA.CONFIG_FP_DISABLE )
   END_RUNG wire#w1
   // the same network as SCL:
   IF #STATIC_DATA.CONFIG_SIM_DISABLE OR #STATIC_DATA.CONFIG_FP_DISABLE THEN
       #DYNAMIC_DATA.mode_SimOn := FALSE;
   END_IF;
END_REGION

REGION Network 7: Signal Conditioning — Remote/local modes disabled
   // ▀▀▀▀▀▀▀▀▀▀▀▀▀▀▀▀▀▀▀▀▀▀▀▀▀▀▀▀▀▀▀▀▀▀▀▀▀▀▀▀▀▀▀▀
   // If remote/local mode is not enabled (CONFIG_RL_ENABLE = 0), or if the faceplate is disabled 
   // (CONFIG_FP_DISABLE = 1),reset both mode_RemoteOn and mode_LocalOn.
   // ▄▄▄▄▄▄▄▄▄▄▄▄▄▄▄▄▄▄▄▄▄▄▄▄▄▄▄▄▄▄▄▄▄▄▄▄▄▄▄▄▄▄▄▄
   RUNG wire#powerrail
      I_Contact( #STATIC_DATA.CONFIG_RL_ENABLE )
      wire#w1
      R_Coil( #DYNAMIC_DATA.mode_RemoteOn )
   END_RUNG
   RUNG wire#powerrail
      Contact( #STATIC_DATA.CONFIG_FP_DISABLE )
   END_RUNG wire#w1
   RUNG wire#w1
      R_Coil( #DYNAMIC_DATA.mode_LocalOn )
   END_RUNG
   // the same network as SCL:
   IF NOT #STATIC_DATA.CONFIG_RL_ENABLE OR #STATIC_DATA.CONFIG_FP_DISABLE THEN
       #DYNAMIC_DATA.mode_RemoteOn := FALSE;
       #DYNAMIC_DATA.mode_LocalOn := FALSE;
   END_IF;
END_REGION

REGION Network 8: Signal Conditioning — Remote/Local selection if enabled
   // ▀▀▀▀▀▀▀▀▀▀▀▀▀▀▀▀▀▀▀▀▀▀▀▀▀▀▀▀▀▀▀▀▀▀▀▀▀▀▀▀▀▀▀▀
   // If remote/local mode is enabled (CONFIG_RL_ENABLE = 1), and the  faceplate is not disabled 
   // (CONFIG_FP_DISABLE = 0), and:
   // 
   //    1.  Neither mode_RemoteOn or mode_LocalOn is active, default to remote mode
   //    2.  A rising edge is detected on mode_LocalOn, reset mode_RemoteOn (in local)
   //    3.  A rising edge is detected on mode_RemoteOn, reset mode_LocalOn (in remote)
   //    4.  Both mode_RemoteOn and mode_LocalOn is active, default to remote mode
   // ▄▄▄▄▄▄▄▄▄▄▄▄▄▄▄▄▄▄▄▄▄▄▄▄▄▄▄▄▄▄▄▄▄▄▄▄▄▄▄▄▄▄▄▄
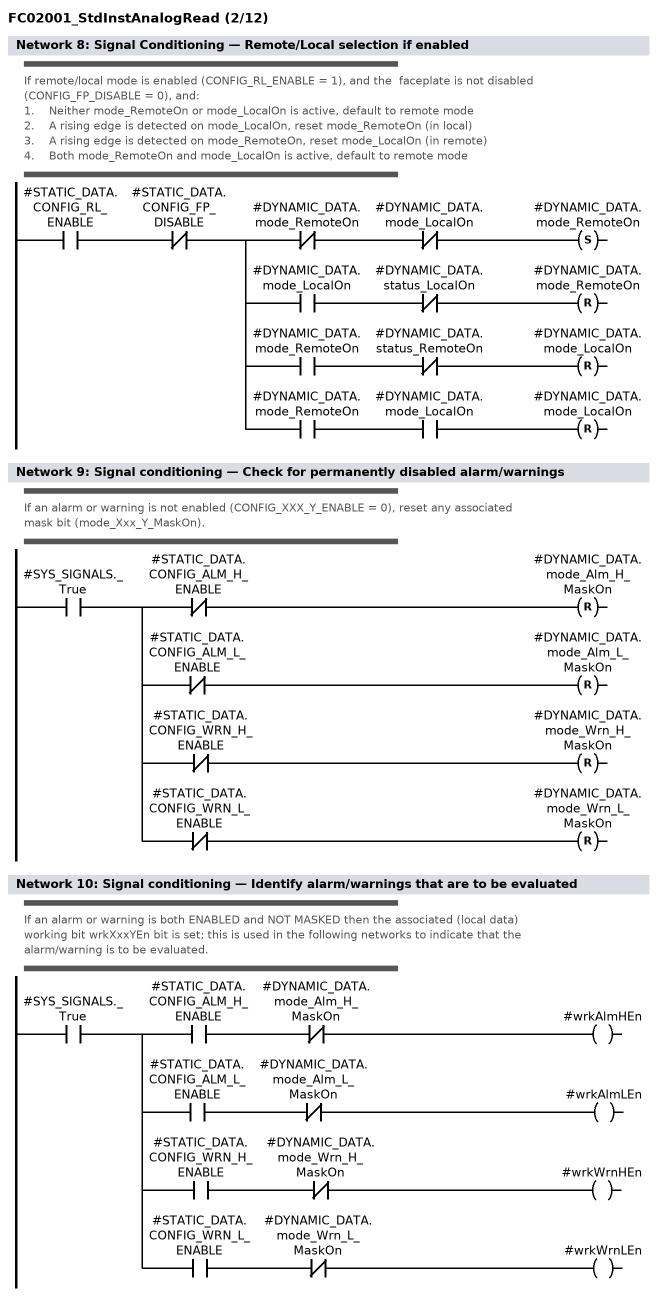
   RUNG wire#powerrail
      Contact( #STATIC_DATA.CONFIG_RL_ENABLE )
      I_Contact( #STATIC_DATA.CONFIG_FP_DISABLE )
      wire#w1
      I_Contact( #DYNAMIC_DATA.mode_RemoteOn )
      I_Contact( #DYNAMIC_DATA.mode_LocalOn )
      S_Coil( #DYNAMIC_DATA.mode_RemoteOn )
   END_RUNG
   RUNG wire#w1
      Contact( #DYNAMIC_DATA.mode_LocalOn )
      I_Contact( #DYNAMIC_DATA.status_LocalOn )
      R_Coil( #DYNAMIC_DATA.mode_RemoteOn )
   END_RUNG
   RUNG wire#w1
      Contact( #DYNAMIC_DATA.mode_RemoteOn )
      I_Contact( #DYNAMIC_DATA.status_RemoteOn )
      R_Coil( #DYNAMIC_DATA.mode_LocalOn )
   END_RUNG
   RUNG wire#w1
      Contact( #DYNAMIC_DATA.mode_RemoteOn )
      Contact( #DYNAMIC_DATA.mode_LocalOn )
      R_Coil( #DYNAMIC_DATA.mode_LocalOn )
   END_RUNG
   // the same network as SCL:
   #_w1 := #STATIC_DATA.CONFIG_RL_ENABLE AND NOT #STATIC_DATA.CONFIG_FP_DISABLE;
   IF #_w1 AND NOT #DYNAMIC_DATA.mode_RemoteOn AND NOT #DYNAMIC_DATA.mode_LocalOn THEN
       #DYNAMIC_DATA.mode_RemoteOn := TRUE;
   END_IF;
   IF #_w1 AND #DYNAMIC_DATA.mode_LocalOn AND NOT #DYNAMIC_DATA.status_LocalOn THEN
       #DYNAMIC_DATA.mode_RemoteOn := FALSE;
   END_IF;
   IF #_w1 AND #DYNAMIC_DATA.mode_RemoteOn AND NOT #DYNAMIC_DATA.status_RemoteOn THEN
       #DYNAMIC_DATA.mode_LocalOn := FALSE;
   END_IF;
   IF #_w1 AND #DYNAMIC_DATA.mode_RemoteOn AND #DYNAMIC_DATA.mode_LocalOn THEN
       #DYNAMIC_DATA.mode_LocalOn := FALSE;
   END_IF;
END_REGION

REGION Network 9: Signal conditioning — Check for permanently disabled alarm/warnings
   // ▀▀▀▀▀▀▀▀▀▀▀▀▀▀▀▀▀▀▀▀▀▀▀▀▀▀▀▀▀▀▀▀▀▀▀▀▀▀▀▀▀▀▀▀
   // If an alarm or warning is not enabled (CONFIG_XXX_Y_ENABLE = 0), reset any associated 
   // mask bit (mode_Xxx_Y_MaskOn).
   // ▄▄▄▄▄▄▄▄▄▄▄▄▄▄▄▄▄▄▄▄▄▄▄▄▄▄▄▄▄▄▄▄▄▄▄▄▄▄▄▄▄▄▄▄
   RUNG wire#powerrail
      Contact( #SYS_SIGNALS._True )
      wire#w1
      I_Contact( #STATIC_DATA.CONFIG_ALM_H_ENABLE )
      R_Coil( #DYNAMIC_DATA.mode_Alm_H_MaskOn )
   END_RUNG
   RUNG wire#w1
      I_Contact( #STATIC_DATA.CONFIG_ALM_L_ENABLE )
      R_Coil( #DYNAMIC_DATA.mode_Alm_L_MaskOn )
   END_RUNG
   RUNG wire#w1
      I_Contact( #STATIC_DATA.CONFIG_WRN_H_ENABLE )
      R_Coil( #DYNAMIC_DATA.mode_Wrn_H_MaskOn )
   END_RUNG
   RUNG wire#w1
      I_Contact( #STATIC_DATA.CONFIG_WRN_L_ENABLE )
      R_Coil( #DYNAMIC_DATA.mode_Wrn_L_MaskOn )
   END_RUNG
   // the same network as SCL:
   IF #SYS_SIGNALS._True AND NOT #STATIC_DATA.CONFIG_ALM_H_ENABLE THEN
       #DYNAMIC_DATA.mode_Alm_H_MaskOn := FALSE;
   END_IF;
   IF #SYS_SIGNALS._True AND NOT #STATIC_DATA.CONFIG_ALM_L_ENABLE THEN
       #DYNAMIC_DATA.mode_Alm_L_MaskOn := FALSE;
   END_IF;
   IF #SYS_SIGNALS._True AND NOT #STATIC_DATA.CONFIG_WRN_H_ENABLE THEN
       #DYNAMIC_DATA.mode_Wrn_H_MaskOn := FALSE;
   END_IF;
   IF #SYS_SIGNALS._True AND NOT #STATIC_DATA.CONFIG_WRN_L_ENABLE THEN
       #DYNAMIC_DATA.mode_Wrn_L_MaskOn := FALSE;
   END_IF;
END_REGION

REGION Network 10: Signal conditioning — Identify alarm/warnings that are to be evaluated
   // ▀▀▀▀▀▀▀▀▀▀▀▀▀▀▀▀▀▀▀▀▀▀▀▀▀▀▀▀▀▀▀▀▀▀▀▀▀▀▀▀▀▀▀▀
   // If an alarm or warning is both ENABLED and NOT MASKED then the associated (local data) 
   // working bit wrkXxxYEn bit is set; this is used in the following networks to indicate that the 
   // alarm/warning is to be evaluated.
   // ▄▄▄▄▄▄▄▄▄▄▄▄▄▄▄▄▄▄▄▄▄▄▄▄▄▄▄▄▄▄▄▄▄▄▄▄▄▄▄▄▄▄▄▄
   RUNG wire#powerrail
      Contact( #SYS_SIGNALS._True )
      wire#w1
      Contact( #STATIC_DATA.CONFIG_ALM_H_ENABLE )
      I_Contact( #DYNAMIC_DATA.mode_Alm_H_MaskOn )
      Coil( #wrkAlmHEn )
   END_RUNG
   RUNG wire#w1
      Contact( #STATIC_DATA.CONFIG_ALM_L_ENABLE )
      I_Contact( #DYNAMIC_DATA.mode_Alm_L_MaskOn )
      Coil( #wrkAlmLEn )
   END_RUNG
   RUNG wire#w1
      Contact( #STATIC_DATA.CONFIG_WRN_H_ENABLE )
      I_Contact( #DYNAMIC_DATA.mode_Wrn_H_MaskOn )
      Coil( #wrkWrnHEn )
   END_RUNG
   RUNG wire#w1
      Contact( #STATIC_DATA.CONFIG_WRN_L_ENABLE )
      I_Contact( #DYNAMIC_DATA.mode_Wrn_L_MaskOn )
      Coil( #wrkWrnLEn )
   END_RUNG
   // the same network as SCL:
   #wrkAlmHEn := #SYS_SIGNALS._True AND #STATIC_DATA.CONFIG_ALM_H_ENABLE AND NOT #DYNAMIC_DATA.mode_Alm_H_MaskOn;
   #wrkAlmLEn := #SYS_SIGNALS._True AND #STATIC_DATA.CONFIG_ALM_L_ENABLE AND NOT #DYNAMIC_DATA.mode_Alm_L_MaskOn;
   #wrkWrnHEn := #SYS_SIGNALS._True AND #STATIC_DATA.CONFIG_WRN_H_ENABLE AND NOT #DYNAMIC_DATA.mode_Wrn_H_MaskOn;
   #wrkWrnLEn := #SYS_SIGNALS._True AND #STATIC_DATA.CONFIG_WRN_L_ENABLE AND NOT #DYNAMIC_DATA.mode_Wrn_L_MaskOn;
END_REGION

REGION Network 11: Signal conditioning — Reset the data for alarm/warnings that are not enabled
   // ▀▀▀▀▀▀▀▀▀▀▀▀▀▀▀▀▀▀▀▀▀▀▀▀▀▀▀▀▀▀▀▀▀▀▀▀▀▀▀▀▀▀▀▀
   // If an alarm or warning is not enabled or is masked (indicated by wrkXxxYEn = 0), the associated 
   // message bit (msg_Xxx_Y) for the alarm or warning is permanently deactivated (reset).
   // 
   // Similarly, the associated actual timer for the alarm or warning (actual_Xxx_Y_Timer) is set to 
   // zero.
   // ▄▄▄▄▄▄▄▄▄▄▄▄▄▄▄▄▄▄▄▄▄▄▄▄▄▄▄▄▄▄▄▄▄▄▄▄▄▄▄▄▄▄▄▄
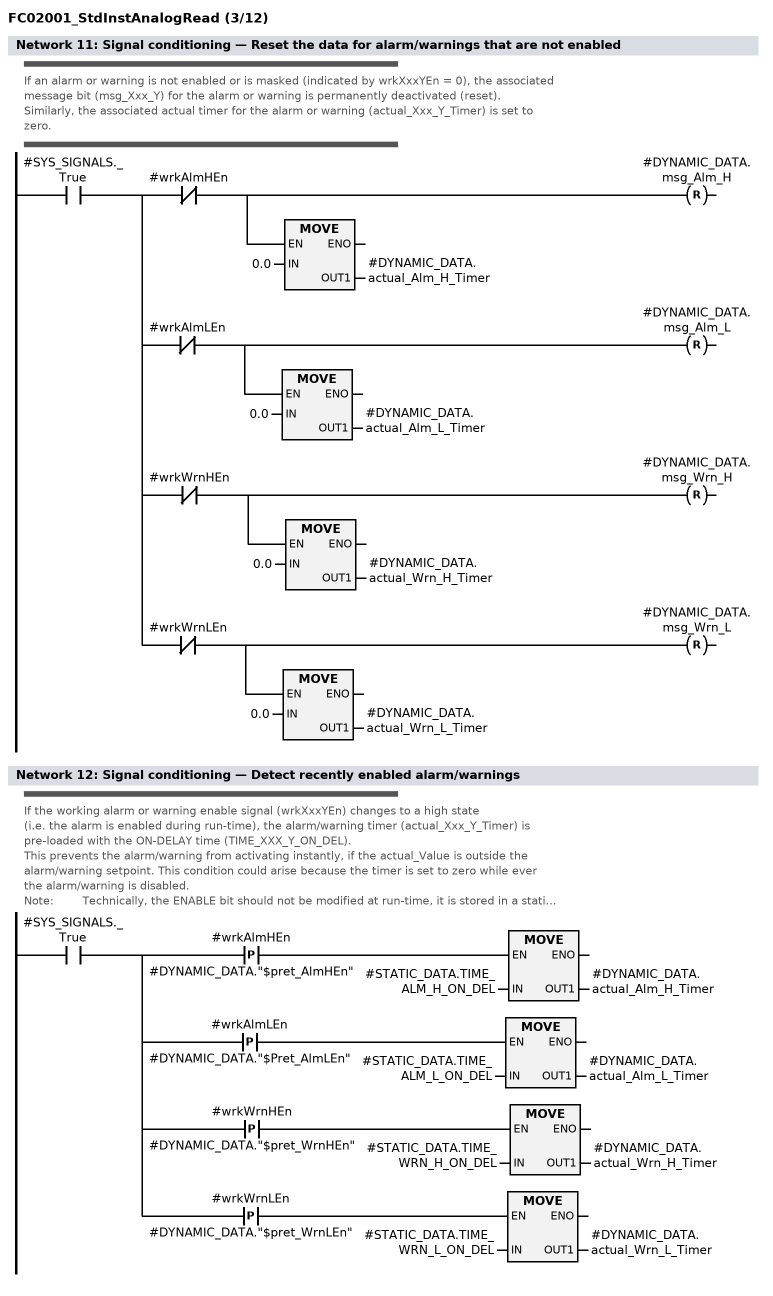
   RUNG wire#powerrail
      Contact( #SYS_SIGNALS._True )
      wire#w1
      I_Contact( #wrkAlmHEn )
      wire#w2
      R_Coil( #DYNAMIC_DATA.msg_Alm_H )
   END_RUNG
   RUNG wire#w2
      { S7_GenerateENO := "TRUE" } Move(in := 0.0, out1 => #DYNAMIC_DATA.actual_Alm_H_Timer)
   END_RUNG
   RUNG wire#w1
      I_Contact( #wrkAlmLEn )
      wire#w3
      R_Coil( #DYNAMIC_DATA.msg_Alm_L )
   END_RUNG
   RUNG wire#w3
      { S7_GenerateENO := "TRUE" } Move(in := 0.0, out1 => #DYNAMIC_DATA.actual_Alm_L_Timer)
   END_RUNG
   RUNG wire#w1
      I_Contact( #wrkWrnHEn )
      wire#w4
      R_Coil( #DYNAMIC_DATA.msg_Wrn_H )
   END_RUNG
   RUNG wire#w4
      { S7_GenerateENO := "TRUE" } Move(in := 0.0, out1 => #DYNAMIC_DATA.actual_Wrn_H_Timer)
   END_RUNG
   RUNG wire#w1
      I_Contact( #wrkWrnLEn )
      wire#w5
      R_Coil( #DYNAMIC_DATA.msg_Wrn_L )
   END_RUNG
   RUNG wire#w5
      { S7_GenerateENO := "TRUE" } Move(in := 0.0, out1 => #DYNAMIC_DATA.actual_Wrn_L_Timer)
   END_RUNG
   // the same network as SCL:
   IF #SYS_SIGNALS._True AND NOT #wrkAlmHEn THEN
       #DYNAMIC_DATA.msg_Alm_H := FALSE;
       #DYNAMIC_DATA.actual_Alm_H_Timer := 0.0;
   END_IF;
   IF #SYS_SIGNALS._True AND NOT #wrkAlmLEn THEN
       #DYNAMIC_DATA.msg_Alm_L := FALSE;
       #DYNAMIC_DATA.actual_Alm_L_Timer := 0.0;
   END_IF;
   IF #SYS_SIGNALS._True AND NOT #wrkWrnHEn THEN
       #DYNAMIC_DATA.msg_Wrn_H := FALSE;
       #DYNAMIC_DATA.actual_Wrn_H_Timer := 0.0;
   END_IF;
   IF #SYS_SIGNALS._True AND NOT #wrkWrnLEn THEN
       #DYNAMIC_DATA.msg_Wrn_L := FALSE;
       #DYNAMIC_DATA.actual_Wrn_L_Timer := 0.0;
   END_IF;
END_REGION

REGION Network 12: Signal conditioning — Detect recently enabled alarm/warnings
   // ▀▀▀▀▀▀▀▀▀▀▀▀▀▀▀▀▀▀▀▀▀▀▀▀▀▀▀▀▀▀▀▀▀▀▀▀▀▀▀▀▀▀▀▀
   // If the working alarm or warning enable signal (wrkXxxYEn) changes to a high state
   // (i.e. the alarm is enabled during run-time), the alarm/warning timer (actual_Xxx_Y_Timer) is 
   // pre-loaded with the ON-DELAY time (TIME_XXX_Y_ON_DEL).
   // 
   // This prevents the alarm/warning from activating instantly, if the actual_Value is outside the
   // alarm/warning setpoint. This condition could arise because the timer is set to zero while ever
   // the alarm/warning is disabled.
   // 
   // Note:    Technically, the ENABLE bit should not be modified at run-time, it is stored in a static
   //      data block; however, the condition could arise if that static data block is being used
   //      as a recipe block. mask signals can of course be changed at run-time.
   // ▄▄▄▄▄▄▄▄▄▄▄▄▄▄▄▄▄▄▄▄▄▄▄▄▄▄▄▄▄▄▄▄▄▄▄▄▄▄▄▄▄▄▄▄
   RUNG wire#powerrail
      Contact( #SYS_SIGNALS._True )
      wire#w1
      P_Contact(operand := #wrkAlmHEn, bit := #DYNAMIC_DATA."$pret_AlmHEn")
      { S7_GenerateENO := "TRUE" } Move(in := #STATIC_DATA.TIME_ALM_H_ON_DEL, out1 => #DYNAMIC_DATA.actual_Alm_H_Timer)
   END_RUNG
   RUNG wire#w1
      P_Contact(operand := #wrkAlmLEn, bit := #DYNAMIC_DATA."$Pret_AlmLEn")
      { S7_GenerateENO := "TRUE" } Move(in := #STATIC_DATA.TIME_ALM_L_ON_DEL, out1 => #DYNAMIC_DATA.actual_Alm_L_Timer)
   END_RUNG
   RUNG wire#w1
      P_Contact(operand := #wrkWrnHEn, bit := #DYNAMIC_DATA."$pret_WrnHEn")
      { S7_GenerateENO := "TRUE" } Move(in := #STATIC_DATA.TIME_WRN_H_ON_DEL, out1 => #DYNAMIC_DATA.actual_Wrn_H_Timer)
   END_RUNG
   RUNG wire#w1
      P_Contact(operand := #wrkWrnLEn, bit := #DYNAMIC_DATA."$pret_WrnLEn")
      { S7_GenerateENO := "TRUE" } Move(in := #STATIC_DATA.TIME_WRN_L_ON_DEL, out1 => #DYNAMIC_DATA.actual_Wrn_L_Timer)
   END_RUNG
   // the same network as SCL:
   #_w1 := #SYS_SIGNALS._True AND #wrkAlmHEn AND NOT #DYNAMIC_DATA."$pret_AlmHEn";   // rising edge of #wrkAlmHEn
   #DYNAMIC_DATA."$pret_AlmHEn" := #wrkAlmHEn;
   IF #_w1 THEN #DYNAMIC_DATA.actual_Alm_H_Timer := #STATIC_DATA.TIME_ALM_H_ON_DEL; END_IF;
   #_w2 := #SYS_SIGNALS._True AND #wrkAlmLEn AND NOT #DYNAMIC_DATA."$Pret_AlmLEn";   // rising edge of #wrkAlmLEn
   #DYNAMIC_DATA."$Pret_AlmLEn" := #wrkAlmLEn;
   IF #_w2 THEN #DYNAMIC_DATA.actual_Alm_L_Timer := #STATIC_DATA.TIME_ALM_L_ON_DEL; END_IF;
   #_w3 := #SYS_SIGNALS._True AND #wrkWrnHEn AND NOT #DYNAMIC_DATA."$pret_WrnHEn";   // rising edge of #wrkWrnHEn
   #DYNAMIC_DATA."$pret_WrnHEn" := #wrkWrnHEn;
   IF #_w3 THEN #DYNAMIC_DATA.actual_Wrn_H_Timer := #STATIC_DATA.TIME_WRN_H_ON_DEL; END_IF;
   #_w4 := #SYS_SIGNALS._True AND #wrkWrnLEn AND NOT #DYNAMIC_DATA."$pret_WrnLEn";   // rising edge of #wrkWrnLEn
   #DYNAMIC_DATA."$pret_WrnLEn" := #wrkWrnLEn;
   IF #_w4 THEN #DYNAMIC_DATA.actual_Wrn_L_Timer := #STATIC_DATA.TIME_WRN_L_ON_DEL; END_IF;
END_REGION

REGION Network 13: Signal conditioning — Ensure Out of Range percentage is 10% or less
   // ▀▀▀▀▀▀▀▀▀▀▀▀▀▀▀▀▀▀▀▀▀▀▀▀▀▀▀▀▀▀▀▀▀▀▀▀▀▀▀▀▀▀▀▀
   // The RANGE_OOR_PERCENT signal is checked to ensure it is within the range 0.0 to 10.0.
   // 
   // The local data wrkOORPercent holds the corrected value and is used in the out of range 
   // calculations
   // ▄▄▄▄▄▄▄▄▄▄▄▄▄▄▄▄▄▄▄▄▄▄▄▄▄▄▄▄▄▄▄▄▄▄▄▄▄▄▄▄▄▄▄▄
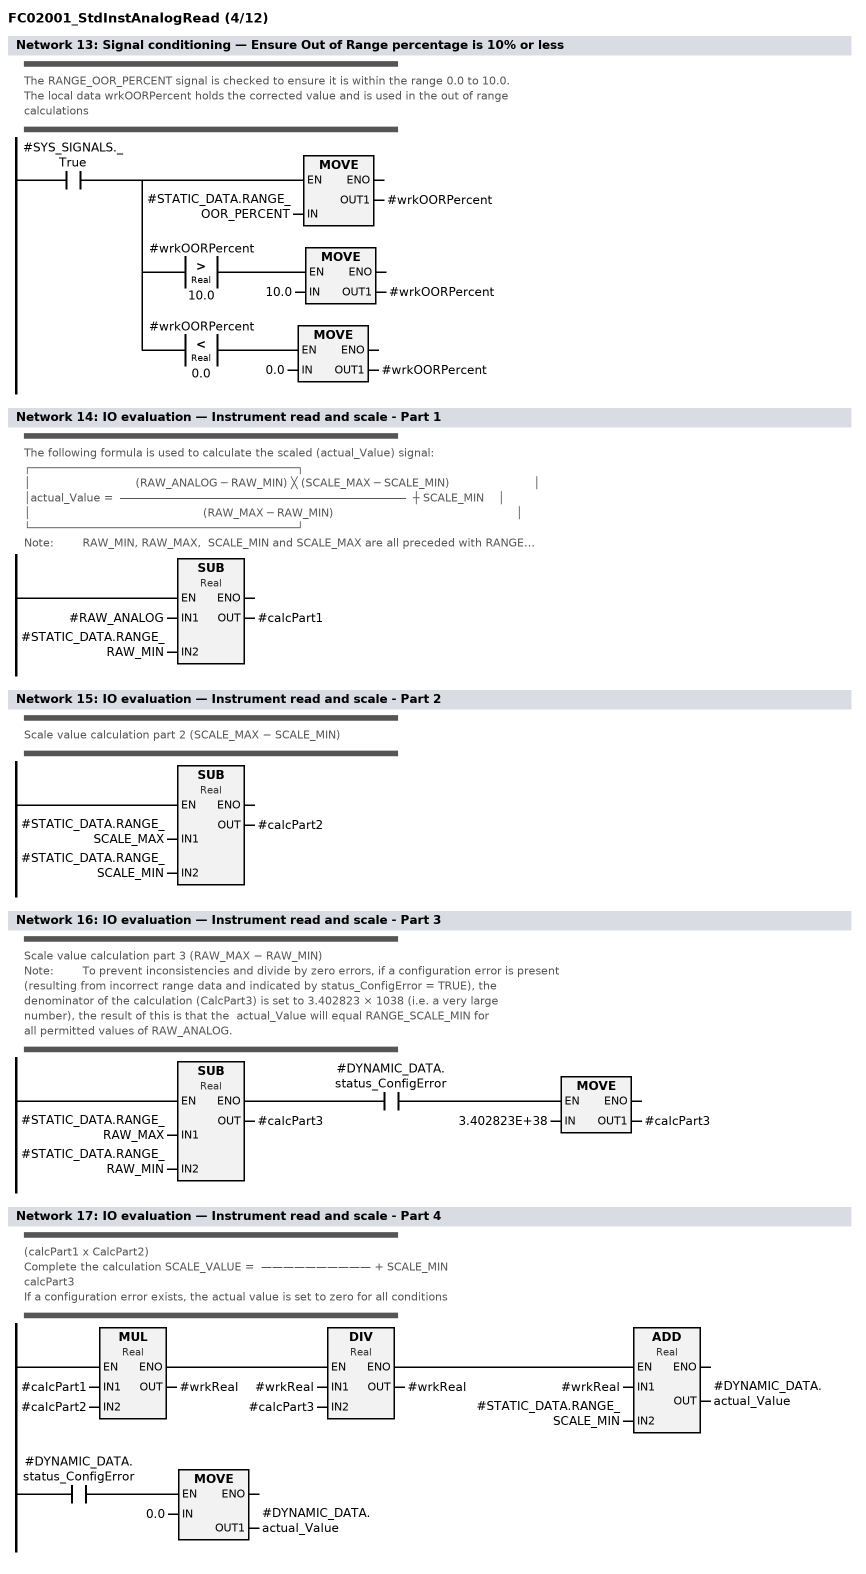
   RUNG wire#powerrail
      Contact( #SYS_SIGNALS._True )
      wire#w1
      { S7_GenerateENO := "TRUE" } Move(in := #STATIC_DATA.RANGE_OOR_PERCENT, out1 => #wrkOORPercent)
   END_RUNG
   RUNG wire#w1
      { S7_Templates := "SrcType := Real" } GT_Contact(in1 := #wrkOORPercent, in2 := 10.0)
      { S7_GenerateENO := "TRUE" } Move(in := 10.0, out1 => #wrkOORPercent)
   END_RUNG
   RUNG wire#w1
      { S7_Templates := "SrcType := Real" } LT_Contact(in1 := #wrkOORPercent, in2 := 0.0)
      { S7_GenerateENO := "TRUE" } Move(in := 0.0, out1 => #wrkOORPercent)
   END_RUNG
   // the same network as SCL:
   IF #SYS_SIGNALS._True THEN #wrkOORPercent := #STATIC_DATA.RANGE_OOR_PERCENT; END_IF;
   IF #SYS_SIGNALS._True AND (#wrkOORPercent > 10.0) THEN #wrkOORPercent := 10.0; END_IF;
   IF #SYS_SIGNALS._True AND (#wrkOORPercent < 0.0) THEN #wrkOORPercent := 0.0; END_IF;
END_REGION

REGION Network 14: IO evaluation — Instrument read and scale - Part 1
   // ▀▀▀▀▀▀▀▀▀▀▀▀▀▀▀▀▀▀▀▀▀▀▀▀▀▀▀▀▀▀▀▀▀▀▀▀▀▀▀▀▀▀▀▀
   // The following formula is used to calculate the scaled (actual_Value) signal:
   // ┌─────────────────────────────────────────┐
   // │                              (RAW_ANALOG ─ RAW_MIN) ╳ (SCALE_MAX ─ SCALE_MIN)            │
   // │actual_Value =  ――――――――――――――――――――――――――  ┼ SCALE_MIN    │
   // │                              (RAW_MAX ─ RAW_MIN)                    │
   // └─────────────────────────────────────────┘
   // Note:    RAW_MIN, RAW_MAX,  SCALE_MIN and SCALE_MAX are all preceded with RANGE_
   //      in the above equation 
   // 
   // Scale value calculation part 1 is (RAW_ANALOG − RAW_MIN)
   // ▄▄▄▄▄▄▄▄▄▄▄▄▄▄▄▄▄▄▄▄▄▄▄▄▄▄▄▄▄▄▄▄▄▄▄▄▄▄▄▄▄▄▄▄
   RUNG wire#powerrail
      { S7_Templates := "SrcType := Real"; S7_GenerateENO := "TRUE" } Sub(in1 := #RAW_ANALOG, in2 := #STATIC_DATA.RANGE_RAW_MIN, out => #calcPart1)
   END_RUNG
   // the same network as SCL:
   #calcPart1 := #RAW_ANALOG - #STATIC_DATA.RANGE_RAW_MIN;
END_REGION

